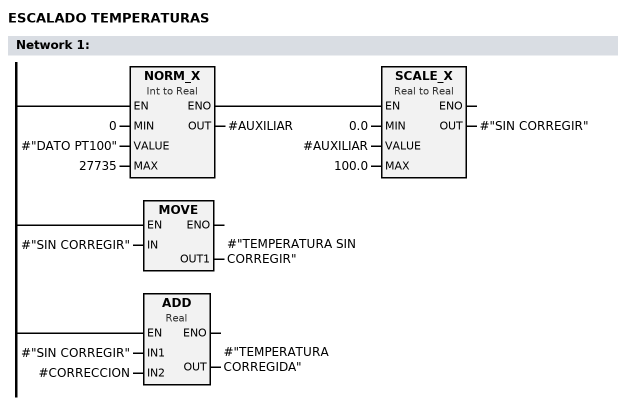
   RUNG wire#powerrail
      { S7_Templates := "[SrcType := Int, DestType := Real]" } Normalize(min := 0, value := #"DATO PT100", max := 27735, out => #AUXILIAR)
      { S7_Templates := "[SrcType := Real, DestType := Real]" } Scale(min := 0.0, value := #AUXILIAR, max := 100.0, out => #"SIN CORREGIR")
   END_RUNG
   RUNG wire#powerrail
      Move(in := #"SIN CORREGIR", out1 => #"TEMPERATURA SIN CORREGIR")
   END_RUNG
   RUNG wire#powerrail
      { S7_Templates := "SrcType := Real" } Add(in1 := #"SIN CORREGIR", in2 := #CORRECCION, out => #"TEMPERATURA CORREGIDA")
   END_RUNG
   // the same network as SCL:
   #AUXILIAR := NORM_X(MIN := 0, VALUE := #"DATO PT100", MAX := 27735);
   #"SIN CORREGIR" := SCALE_X(MIN := 0.0, VALUE := #AUXILIAR, MAX := 100.0);
   #"TEMPERATURA SIN CORREGIR" := #"SIN CORREGIR";
   #"TEMPERATURA CORREGIDA" := #"SIN CORREGIR" + #CORRECCION;
END_REGION
END_FUNCTION

FUNCTION "CONVERSOR MIN A MS" : Void   // FC2, LAD
{ S7_Optimized_Access := 'TRUE' }
VERSION : 0.1
   VAR_INPUT
      "TIEMPO EN MIN" : Int;
   END_VAR
   VAR_OUTPUT
      "TIEMPO EN MS" : DInt;
   END_VAR
BEGIN

REGION Network 1
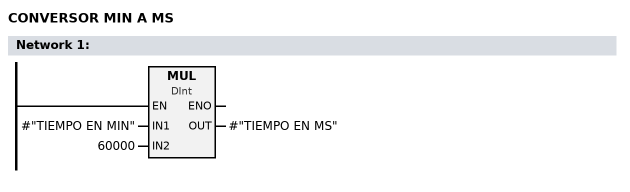
   RUNG wire#powerrail
      { S7_Templates := "SrcType := DInt" } Mul(in1 := #"TIEMPO EN MIN", in2 := 60000, out => #"TIEMPO EN MS")
   END_RUNG
   // the same network as SCL:
   #"TIEMPO EN MS" := #"TIEMPO EN MIN" * 60000;
END_REGION
END_FUNCTION

FUNCTION "CONVERSOR MS A MIN" : Void   // FC3, LAD
{ S7_Optimized_Access := 'TRUE' }
VERSION : 0.1
   VAR_INPUT
      "TIEMPO EN MS" : DInt;
   END_VAR
   VAR_OUTPUT
      "TIEMPO EN MIN" : Int;
   END_VAR
BEGIN

REGION Network 1
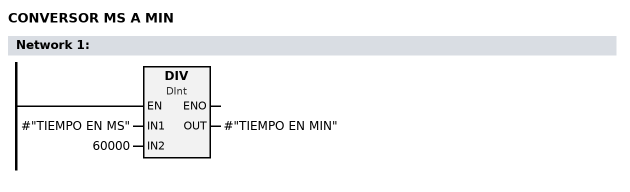
   RUNG wire#powerrail
      { S7_Templates := "SrcType := DInt" } Div(in1 := #"TIEMPO EN MS", in2 := 60000, out => #"TIEMPO EN MIN")
   END_RUNG
   // the same network as SCL:
   #"TIEMPO EN MIN" := #"TIEMPO EN MS" / 60000;
END_REGION
END_FUNCTION

ORGANIZATION_BLOCK "Main"   // OB1, LAD, ProgramCycle
TITLE = "Main Program Sweep (Cycle)"
{ S7_Optimized_Access := 'TRUE' }
VERSION : 0.1
   VAR_INPUT
      Initial_Call : Bool;   // Initial call of this OB
      Remanence : Bool;   // =True, if remanent data are available
   END_VAR
   VAR CONSTANT
      "LARGO REGLA" : Int := 1240;
      COCINA : String := 'COCINA';
      ENFRIADOR : String := 'ENFRIADOR';
   END_VAR
   VAR_TEMP   // added for the SCL form of the ladder/FBD networks
      _w1 : Bool;
   END_VAR
BEGIN

REGION Network 1: REARME
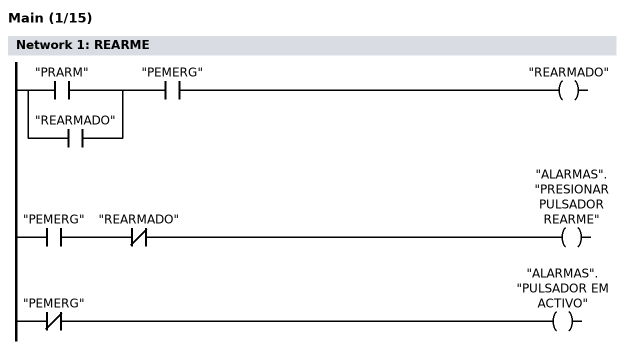
   RUNG wire#powerrail
      Contact( "PRARM" )
      wire#w1
      Contact( "PEMERG" )
      Coil( "REARMADO" )
   END_RUNG
   RUNG wire#powerrail
      Contact( "REARMADO" )
   END_RUNG wire#w1
   RUNG wire#powerrail
      Contact( "PEMERG" )
      I_Contact( "REARMADO" )
      Coil( "ALARMAS"."PRESIONAR PULSADOR REARME" )
   END_RUNG
   RUNG wire#powerrail
      I_Contact( "PEMERG" )
      Coil( "ALARMAS"."PULSADOR EM ACTIVO" )
   END_RUNG
   // the same network as SCL:
   "REARMADO" := ("PRARM" OR "REARMADO") AND "PEMERG";
   "ALARMAS"."PRESIONAR PULSADOR REARME" := "PEMERG" AND NOT "REARMADO";
   "ALARMAS"."PULSADOR EM ACTIVO" := NOT "PEMERG";
END_REGION

REGION Network 2: SELECCION DE NUMERO DE EQUIPO
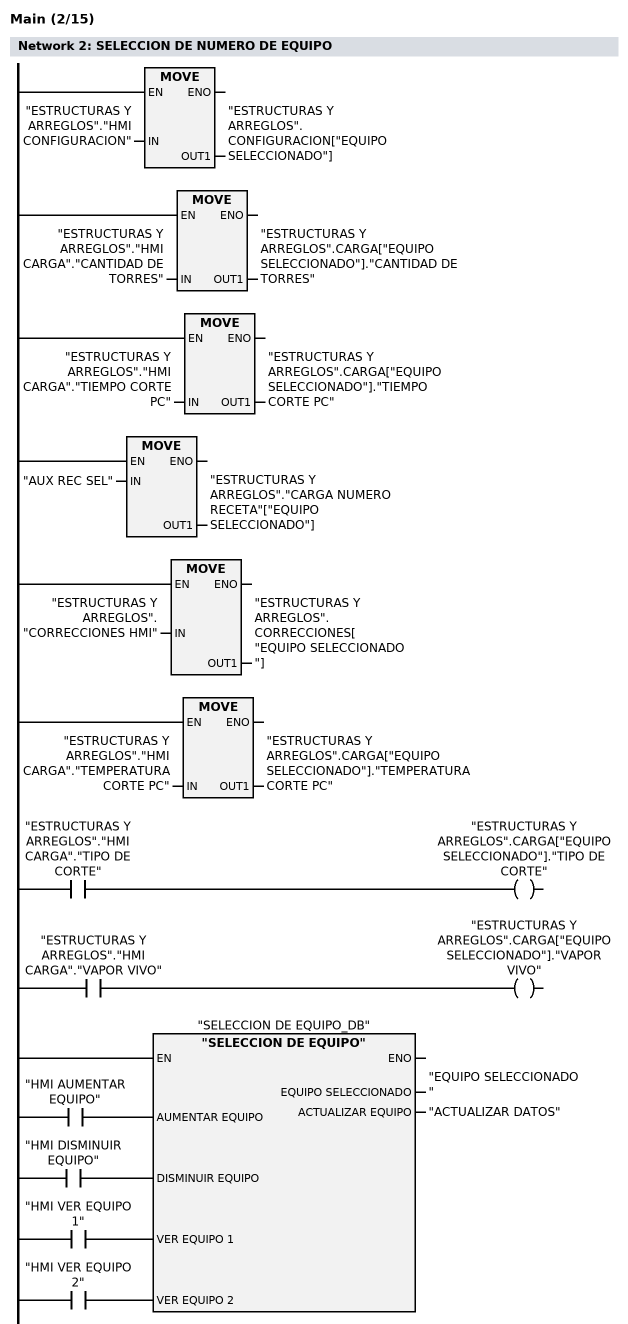
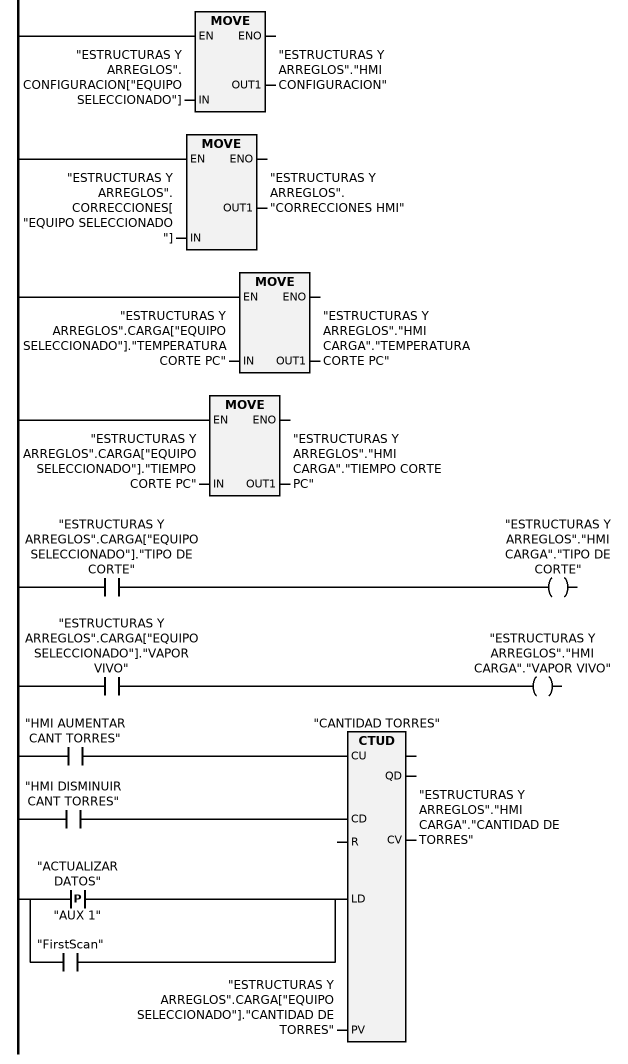
   "ESTRUCTURAS Y ARREGLOS".CONFIGURACION["EQUIPO SELECCIONADO"] := "ESTRUCTURAS Y ARREGLOS"."HMI CONFIGURACION";
   "ESTRUCTURAS Y ARREGLOS".CARGA["EQUIPO SELECCIONADO"]."CANTIDAD DE TORRES" := "ESTRUCTURAS Y ARREGLOS"."HMI CARGA"."CANTIDAD DE TORRES";
   "ESTRUCTURAS Y ARREGLOS".CARGA["EQUIPO SELECCIONADO"]."TIEMPO CORTE PC" := "ESTRUCTURAS Y ARREGLOS"."HMI CARGA"."TIEMPO CORTE PC";
   "ESTRUCTURAS Y ARREGLOS"."CARGA NUMERO RECETA"["EQUIPO SELECCIONADO"] := "AUX REC SEL";
   "ESTRUCTURAS Y ARREGLOS".CORRECCIONES["EQUIPO SELECCIONADO"] := "ESTRUCTURAS Y ARREGLOS"."CORRECCIONES HMI";
   "ESTRUCTURAS Y ARREGLOS".CARGA["EQUIPO SELECCIONADO"]."TEMPERATURA CORTE PC" := "ESTRUCTURAS Y ARREGLOS"."HMI CARGA"."TEMPERATURA CORTE PC";
   "ESTRUCTURAS Y ARREGLOS".CARGA["EQUIPO SELECCIONADO"]."TIPO DE CORTE" := "ESTRUCTURAS Y ARREGLOS"."HMI CARGA"."TIPO DE CORTE";
   "ESTRUCTURAS Y ARREGLOS".CARGA["EQUIPO SELECCIONADO"]."VAPOR VIVO" := "ESTRUCTURAS Y ARREGLOS"."HMI CARGA"."VAPOR VIVO";
   "SELECCION DE EQUIPO_DB"("AUMENTAR EQUIPO" := "HMI AUMENTAR EQUIPO",   // "SELECCION DE EQUIPO"
                           "DISMINUIR EQUIPO" := "HMI DISMINUIR EQUIPO",
                           "VER EQUIPO 1" := "HMI VER EQUIPO 1",
                           "VER EQUIPO 2" := "HMI VER EQUIPO 2",
                           "EQUIPO SELECCIONADO" => "EQUIPO SELECCIONADO",
                           "ACTUALIZAR EQUIPO" => "ACTUALIZAR DATOS");
   "ESTRUCTURAS Y ARREGLOS"."HMI CONFIGURACION" := "ESTRUCTURAS Y ARREGLOS".CONFIGURACION["EQUIPO SELECCIONADO"];
   "ESTRUCTURAS Y ARREGLOS"."CORRECCIONES HMI" := "ESTRUCTURAS Y ARREGLOS".CORRECCIONES["EQUIPO SELECCIONADO"];
   "ESTRUCTURAS Y ARREGLOS"."HMI CARGA"."TEMPERATURA CORTE PC" := "ESTRUCTURAS Y ARREGLOS".CARGA["EQUIPO SELECCIONADO"]."TEMPERATURA CORTE PC";
   "ESTRUCTURAS Y ARREGLOS"."HMI CARGA"."TIEMPO CORTE PC" := "ESTRUCTURAS Y ARREGLOS".CARGA["EQUIPO SELECCIONADO"]."TIEMPO CORTE PC";
   "ESTRUCTURAS Y ARREGLOS"."HMI CARGA"."TIPO DE CORTE" := "ESTRUCTURAS Y ARREGLOS".CARGA["EQUIPO SELECCIONADO"]."TIPO DE CORTE";
   "ESTRUCTURAS Y ARREGLOS"."HMI CARGA"."VAPOR VIVO" := "ESTRUCTURAS Y ARREGLOS".CARGA["EQUIPO SELECCIONADO"]."VAPOR VIVO";
   #_w1 := "ACTUALIZAR DATOS" AND NOT "AUX 1";   // rising edge of "ACTUALIZAR DATOS"
   "AUX 1" := "ACTUALIZAR DATOS";
   "CANTIDAD TORRES".CTUD(CU := "HMI AUMENTAR CANT TORRES",
                          CD := "HMI DISMINUIR CANT TORRES",
                          LD := #_w1 OR "FirstScan",
                          PV := "ESTRUCTURAS Y ARREGLOS".CARGA["EQUIPO SELECCIONADO"]."CANTIDAD DE TORRES",
                          CV => "ESTRUCTURAS Y ARREGLOS"."HMI CARGA"."CANTIDAD DE TORRES");
END_REGION

REGION Network 3: VISUALIZACION LIMITE CANTIDAD DE EQUIPOS Y CANTIDAD DE TORRES
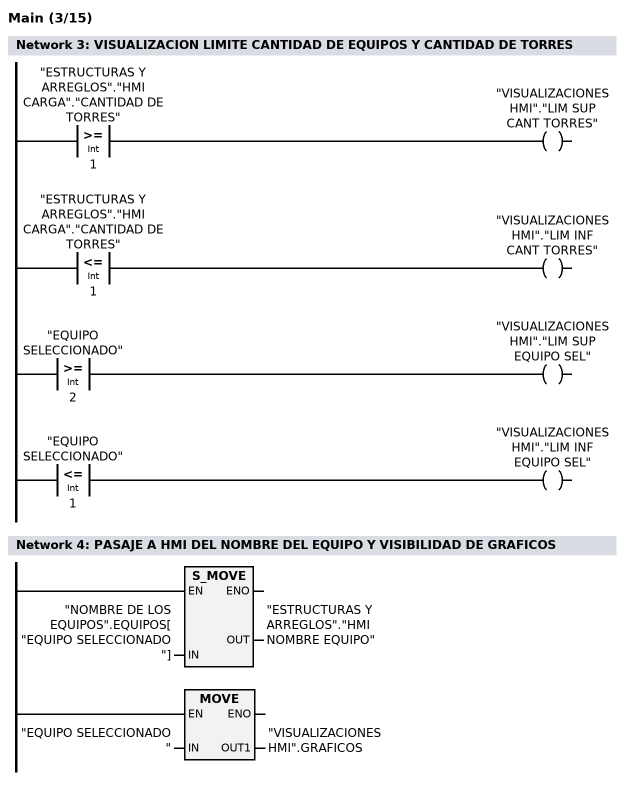
   RUNG wire#powerrail
      { S7_Templates := "SrcType := Int" } GE_Contact(in1 := "ESTRUCTURAS Y ARREGLOS"."HMI CARGA"."CANTIDAD DE TORRES", in2 := 1)
      Coil( "VISUALIZACIONES HMI"."LIM SUP CANT TORRES" )
   END_RUNG
   RUNG wire#powerrail
      { S7_Templates := "SrcType := Int" } LE_Contact(in1 := "ESTRUCTURAS Y ARREGLOS"."HMI CARGA"."CANTIDAD DE TORRES", in2 := 1)
      Coil( "VISUALIZACIONES HMI"."LIM INF CANT TORRES" )
   END_RUNG
   RUNG wire#powerrail
      { S7_Templates := "SrcType := Int" } GE_Contact(in1 := "EQUIPO SELECCIONADO", in2 := 2)
      Coil( "VISUALIZACIONES HMI"."LIM SUP EQUIPO SEL" )
   END_RUNG
   RUNG wire#powerrail
      { S7_Templates := "SrcType := Int" } LE_Contact(in1 := "EQUIPO SELECCIONADO", in2 := 1)
      Coil( "VISUALIZACIONES HMI"."LIM INF EQUIPO SEL" )
   END_RUNG
   // the same network as SCL:
   "VISUALIZACIONES HMI"."LIM SUP CANT TORRES" := "ESTRUCTURAS Y ARREGLOS"."HMI CARGA"."CANTIDAD DE TORRES" >= 1;
   "VISUALIZACIONES HMI"."LIM INF CANT TORRES" := "ESTRUCTURAS Y ARREGLOS"."HMI CARGA"."CANTIDAD DE TORRES" <= 1;
   "VISUALIZACIONES HMI"."LIM SUP EQUIPO SEL" := "EQUIPO SELECCIONADO" >= 2;
   "VISUALIZACIONES HMI"."LIM INF EQUIPO SEL" := "EQUIPO SELECCIONADO" <= 1;
END_REGION

REGION Network 4: PASAJE A HMI DEL NOMBRE DEL EQUIPO Y VISIBILIDAD DE GRAFICOS
   RUNG wire#powerrail
      S_Move(in := "NOMBRE DE LOS EQUIPOS".EQUIPOS["EQUIPO SELECCIONADO"], out => "ESTRUCTURAS Y ARREGLOS"."HMI NOMBRE EQUIPO")
   END_RUNG
   RUNG wire#powerrail
      Move(in := "EQUIPO SELECCIONADO", out1 => "VISUALIZACIONES HMI".GRAFICOS)
   END_RUNG
   // the same network as SCL:
   "ESTRUCTURAS Y ARREGLOS"."HMI NOMBRE EQUIPO" := "NOMBRE DE LOS EQUIPOS".EQUIPOS["EQUIPO SELECCIONADO"];
   "VISUALIZACIONES HMI".GRAFICOS := "EQUIPO SELECCIONADO";
END_REGION

REGION Network 5: BOTON VISUALIZAR RECETA EN PANTALLA "EQUIPO"
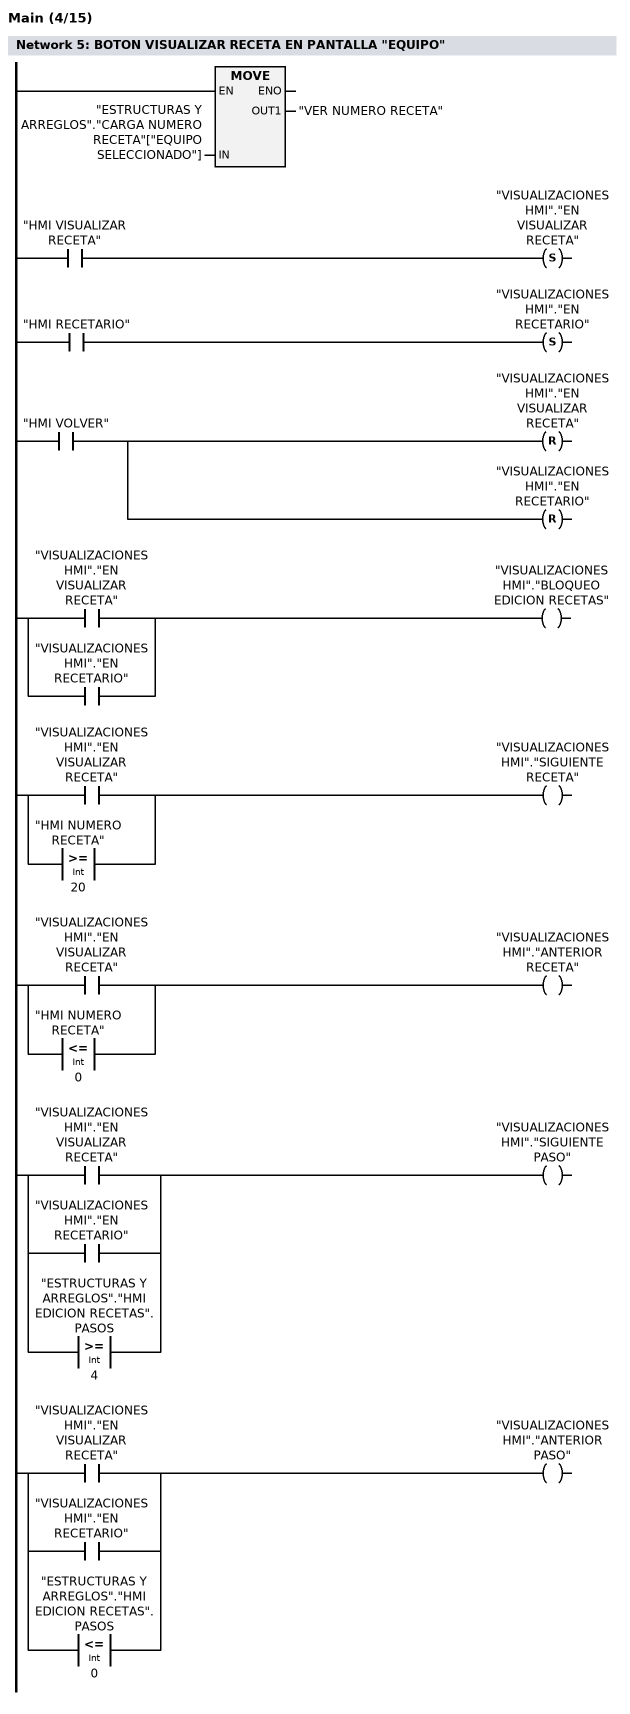
   RUNG wire#powerrail
      Move(in := "ESTRUCTURAS Y ARREGLOS"."CARGA NUMERO RECETA"["EQUIPO SELECCIONADO"], out1 => "VER NUMERO RECETA")
   END_RUNG
   RUNG wire#powerrail
      Contact( "HMI VISUALIZAR RECETA" )
      S_Coil( "VISUALIZACIONES HMI"."EN VISUALIZAR RECETA" )
   END_RUNG
   RUNG wire#powerrail
      Contact( "HMI RECETARIO" )
      S_Coil( "VISUALIZACIONES HMI"."EN RECETARIO" )
   END_RUNG
   RUNG wire#powerrail
      Contact( "HMI VOLVER" )
      wire#w1
      R_Coil( "VISUALIZACIONES HMI"."EN VISUALIZAR RECETA" )
   END_RUNG
   RUNG wire#w1
      R_Coil( "VISUALIZACIONES HMI"."EN RECETARIO" )
   END_RUNG
   RUNG wire#powerrail
      Contact( "VISUALIZACIONES HMI"."EN VISUALIZAR RECETA" )
      wire#w2
      Coil( "VISUALIZACIONES HMI"."BLOQUEO EDICION RECETAS" )
   END_RUNG
   RUNG wire#powerrail
      Contact( "VISUALIZACIONES HMI"."EN RECETARIO" )
   END_RUNG wire#w2
   RUNG wire#powerrail
      Contact( "VISUALIZACIONES HMI"."EN VISUALIZAR RECETA" )
      wire#w3
      Coil( "VISUALIZACIONES HMI"."SIGUIENTE RECETA" )
   END_RUNG
   RUNG wire#powerrail
      { S7_Templates := "SrcType := Int" } GE_Contact(in1 := "HMI NUMERO RECETA", in2 := 20)
   END_RUNG wire#w3
   RUNG wire#powerrail
      Contact( "VISUALIZACIONES HMI"."EN VISUALIZAR RECETA" )
      wire#w4
      Coil( "VISUALIZACIONES HMI"."ANTERIOR RECETA" )
   END_RUNG
   RUNG wire#powerrail
      { S7_Templates := "SrcType := Int" } LE_Contact(in1 := "HMI NUMERO RECETA", in2 := 0)
   END_RUNG wire#w4
   RUNG wire#powerrail
      Contact( "VISUALIZACIONES HMI"."EN VISUALIZAR RECETA" )
      wire#w5
      Coil( "VISUALIZACIONES HMI"."SIGUIENTE PASO" )
   END_RUNG
   RUNG wire#powerrail
      Contact( "VISUALIZACIONES HMI"."EN RECETARIO" )
   END_RUNG wire#w5
   RUNG wire#powerrail
      { S7_Templates := "SrcType := Int" } GE_Contact(in1 := "ESTRUCTURAS Y ARREGLOS"."HMI EDICION RECETAS".PASOS, in2 := 4)
   END_RUNG wire#w5
   RUNG wire#powerrail
      Contact( "VISUALIZACIONES HMI"."EN VISUALIZAR RECETA" )
      wire#w6
      Coil( "VISUALIZACIONES HMI"."ANTERIOR PASO" )
   END_RUNG
   RUNG wire#powerrail
      Contact( "VISUALIZACIONES HMI"."EN RECETARIO" )
   END_RUNG wire#w6
   RUNG wire#powerrail
      { S7_Templates := "SrcType := Int" } LE_Contact(in1 := "ESTRUCTURAS Y ARREGLOS"."HMI EDICION RECETAS".PASOS, in2 := 0)
   END_RUNG wire#w6
   // the same network as SCL:
   "VER NUMERO RECETA" := "ESTRUCTURAS Y ARREGLOS"."CARGA NUMERO RECETA"["EQUIPO SELECCIONADO"];
   IF "HMI VISUALIZAR RECETA" THEN "VISUALIZACIONES HMI"."EN VISUALIZAR RECETA" := TRUE; END_IF;
   IF "HMI RECETARIO" THEN "VISUALIZACIONES HMI"."EN RECETARIO" := TRUE; END_IF;
   IF "HMI VOLVER" THEN
       "VISUALIZACIONES HMI"."EN VISUALIZAR RECETA" := FALSE;
       "VISUALIZACIONES HMI"."EN RECETARIO" := FALSE;
   END_IF;
   "VISUALIZACIONES HMI"."BLOQUEO EDICION RECETAS" := "VISUALIZACIONES HMI"."EN VISUALIZAR RECETA" OR "VISUALIZACIONES HMI"."EN RECETARIO";
   "VISUALIZACIONES HMI"."SIGUIENTE RECETA" := "VISUALIZACIONES HMI"."EN VISUALIZAR RECETA" OR ("HMI NUMERO RECETA" >= 20);
   "VISUALIZACIONES HMI"."ANTERIOR RECETA" := "VISUALIZACIONES HMI"."EN VISUALIZAR RECETA" OR ("HMI NUMERO RECETA" <= 0);
   "VISUALIZACIONES HMI"."SIGUIENTE PASO" := "VISUALIZACIONES HMI"."EN VISUALIZAR RECETA" OR "VISUALIZACIONES HMI"."EN RECETARIO" OR ("ESTRUCTURAS Y ARREGLOS"."HMI EDICION RECETAS".PASOS >= 4);
   "VISUALIZACIONES HMI"."ANTERIOR PASO" := "VISUALIZACIONES HMI"."EN VISUALIZAR RECETA" OR "VISUALIZACIONES HMI"."EN RECETARIO" OR ("ESTRUCTURAS Y ARREGLOS"."HMI EDICION RECETAS".PASOS <= 0);
END_REGION

REGION Network 6: EDITAR RECETAS
   // Receta
   // Recetario
   // Buscar y cargar rece
   // 
   // LOS PASOS TIENE Q IR POR SEPARADOL DE LA ESTRUCTURA
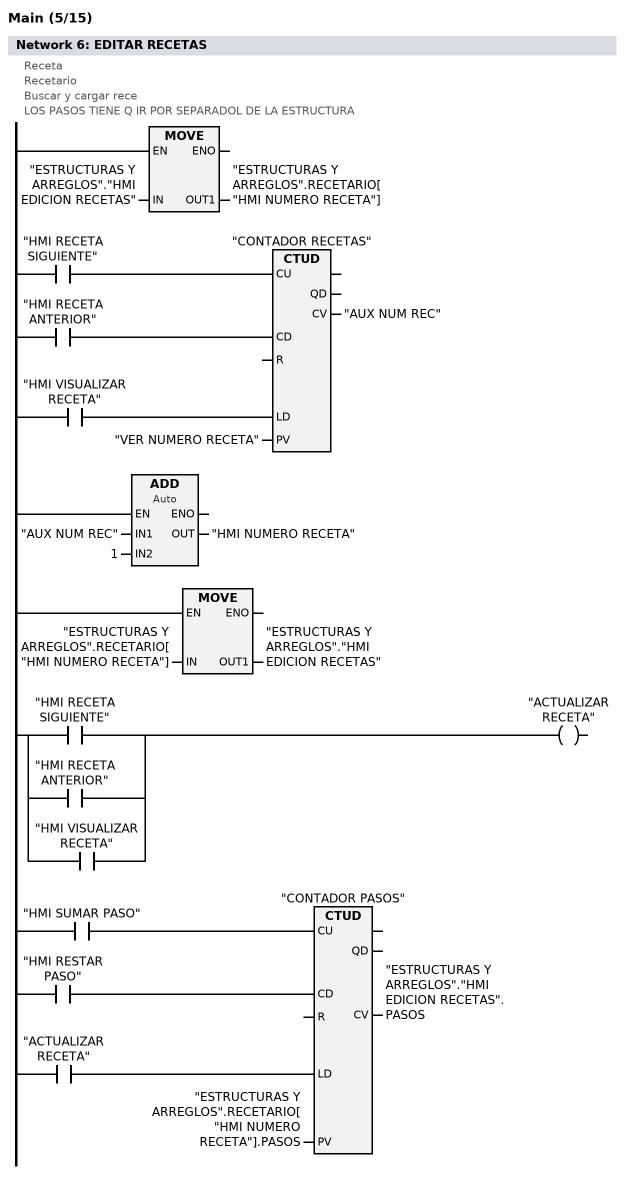
   "ESTRUCTURAS Y ARREGLOS".RECETARIO["HMI NUMERO RECETA"] := "ESTRUCTURAS Y ARREGLOS"."HMI EDICION RECETAS";
   "CONTADOR RECETAS".CTUD(CU := "HMI RECETA SIGUIENTE",
                           CD := "HMI RECETA ANTERIOR",
                           LD := "HMI VISUALIZAR RECETA",
                           PV := "VER NUMERO RECETA",
                           CV => "AUX NUM REC");
   "HMI NUMERO RECETA" := "AUX NUM REC" + 1;
   "ESTRUCTURAS Y ARREGLOS"."HMI EDICION RECETAS" := "ESTRUCTURAS Y ARREGLOS".RECETARIO["HMI NUMERO RECETA"];
   "ACTUALIZAR RECETA" := "HMI RECETA SIGUIENTE" OR "HMI RECETA ANTERIOR" OR "HMI VISUALIZAR RECETA";
   "CONTADOR PASOS".CTUD(CU := "HMI SUMAR PASO",
                         CD := "HMI RESTAR PASO",
                         LD := "ACTUALIZAR RECETA",
                         PV := "ESTRUCTURAS Y ARREGLOS".RECETARIO["HMI NUMERO RECETA"].PASOS,
                         CV => "ESTRUCTURAS Y ARREGLOS"."HMI EDICION RECETAS".PASOS);
END_REGION

REGION Network 7: VISUALIZACIONES RECETA
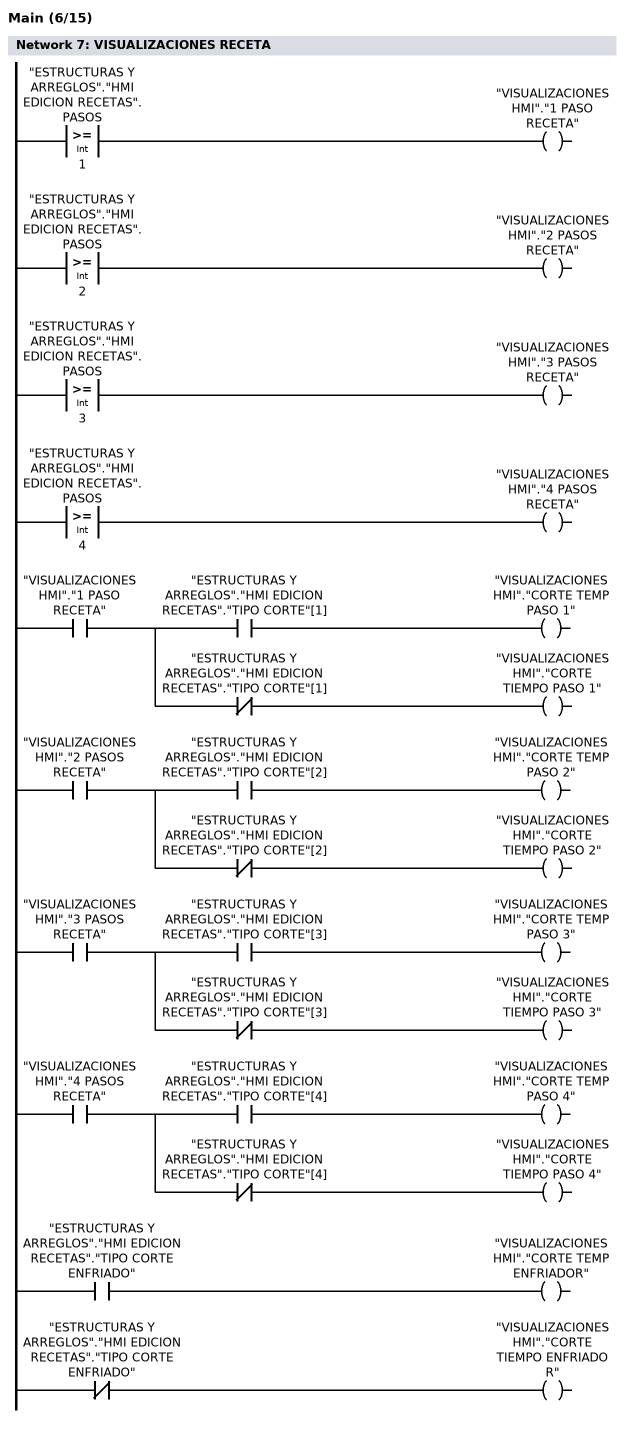
   RUNG wire#powerrail
      { S7_Templates := "SrcType := Int" } GE_Contact(in1 := "ESTRUCTURAS Y ARREGLOS"."HMI EDICION RECETAS".PASOS, in2 := 1)
      Coil( "VISUALIZACIONES HMI"."1 PASO RECETA" )
   END_RUNG
   RUNG wire#powerrail
      { S7_Templates := "SrcType := Int" } GE_Contact(in1 := "ESTRUCTURAS Y ARREGLOS"."HMI EDICION RECETAS".PASOS, in2 := 2)
      Coil( "VISUALIZACIONES HMI"."2 PASOS RECETA" )
   END_RUNG
   RUNG wire#powerrail
      { S7_Templates := "SrcType := Int" } GE_Contact(in1 := "ESTRUCTURAS Y ARREGLOS"."HMI EDICION RECETAS".PASOS, in2 := 3)
      Coil( "VISUALIZACIONES HMI"."3 PASOS RECETA" )
   END_RUNG
   RUNG wire#powerrail
      { S7_Templates := "SrcType := Int" } GE_Contact(in1 := "ESTRUCTURAS Y ARREGLOS"."HMI EDICION RECETAS".PASOS, in2 := 4)
      Coil( "VISUALIZACIONES HMI"."4 PASOS RECETA" )
   END_RUNG
   RUNG wire#powerrail
      Contact( "VISUALIZACIONES HMI"."1 PASO RECETA" )
      wire#w1
      Contact( "ESTRUCTURAS Y ARREGLOS"."HMI EDICION RECETAS"."TIPO CORTE"[1] )
      Coil( "VISUALIZACIONES HMI"."CORTE TEMP PASO 1" )
   END_RUNG
   RUNG wire#w1
      I_Contact( "ESTRUCTURAS Y ARREGLOS"."HMI EDICION RECETAS"."TIPO CORTE"[1] )
      Coil( "VISUALIZACIONES HMI"."CORTE TIEMPO PASO 1" )
   END_RUNG
   RUNG wire#powerrail
      Contact( "VISUALIZACIONES HMI"."2 PASOS RECETA" )
      wire#w2
      Contact( "ESTRUCTURAS Y ARREGLOS"."HMI EDICION RECETAS"."TIPO CORTE"[2] )
      Coil( "VISUALIZACIONES HMI"."CORTE TEMP PASO 2" )
   END_RUNG
   RUNG wire#w2
      I_Contact( "ESTRUCTURAS Y ARREGLOS"."HMI EDICION RECETAS"."TIPO CORTE"[2] )
      Coil( "VISUALIZACIONES HMI"."CORTE TIEMPO PASO 2" )
   END_RUNG
   RUNG wire#powerrail
      Contact( "VISUALIZACIONES HMI"."3 PASOS RECETA" )
      wire#w3
      Contact( "ESTRUCTURAS Y ARREGLOS"."HMI EDICION RECETAS"."TIPO CORTE"[3] )
      Coil( "VISUALIZACIONES HMI"."CORTE TEMP PASO 3" )
   END_RUNG
   RUNG wire#w3
      I_Contact( "ESTRUCTURAS Y ARREGLOS"."HMI EDICION RECETAS"."TIPO CORTE"[3] )
      Coil( "VISUALIZACIONES HMI"."CORTE TIEMPO PASO 3" )
   END_RUNG
   RUNG wire#powerrail
      Contact( "VISUALIZACIONES HMI"."4 PASOS RECETA" )
      wire#w4
      Contact( "ESTRUCTURAS Y ARREGLOS"."HMI EDICION RECETAS"."TIPO CORTE"[4] )
      Coil( "VISUALIZACIONES HMI"."CORTE TEMP PASO 4" )
   END_RUNG
   RUNG wire#w4
      I_Contact( "ESTRUCTURAS Y ARREGLOS"."HMI EDICION RECETAS"."TIPO CORTE"[4] )
      Coil( "VISUALIZACIONES HMI"."CORTE TIEMPO PASO 4" )
   END_RUNG
   RUNG wire#powerrail
      Contact( "ESTRUCTURAS Y ARREGLOS"."HMI EDICION RECETAS"."TIPO CORTE ENFRIADO" )
      Coil( "VISUALIZACIONES HMI"."CORTE TEMP ENFRIADOR" )
   END_RUNG
   RUNG wire#powerrail
      I_Contact( "ESTRUCTURAS Y ARREGLOS"."HMI EDICION RECETAS"."TIPO CORTE ENFRIADO" )
      Coil( "VISUALIZACIONES HMI"."CORTE TIEMPO ENFRIADOR" )
   END_RUNG
   // the same network as SCL:
   "VISUALIZACIONES HMI"."1 PASO RECETA" := "ESTRUCTURAS Y ARREGLOS"."HMI EDICION RECETAS".PASOS >= 1;
   "VISUALIZACIONES HMI"."2 PASOS RECETA" := "ESTRUCTURAS Y ARREGLOS"."HMI EDICION RECETAS".PASOS >= 2;
   "VISUALIZACIONES HMI"."3 PASOS RECETA" := "ESTRUCTURAS Y ARREGLOS"."HMI EDICION RECETAS".PASOS >= 3;
   "VISUALIZACIONES HMI"."4 PASOS RECETA" := "ESTRUCTURAS Y ARREGLOS"."HMI EDICION RECETAS".PASOS >= 4;
   "VISUALIZACIONES HMI"."CORTE TEMP PASO 1" := "VISUALIZACIONES HMI"."1 PASO RECETA" AND "ESTRUCTURAS Y ARREGLOS"."HMI EDICION RECETAS"."TIPO CORTE"[1];
   "VISUALIZACIONES HMI"."CORTE TIEMPO PASO 1" := "VISUALIZACIONES HMI"."1 PASO RECETA" AND NOT "ESTRUCTURAS Y ARREGLOS"."HMI EDICION RECETAS"."TIPO CORTE"[1];
   "VISUALIZACIONES HMI"."CORTE TEMP PASO 2" := "VISUALIZACIONES HMI"."2 PASOS RECETA" AND "ESTRUCTURAS Y ARREGLOS"."HMI EDICION RECETAS"."TIPO CORTE"[2];
   "VISUALIZACIONES HMI"."CORTE TIEMPO PASO 2" := "VISUALIZACIONES HMI"."2 PASOS RECETA" AND NOT "ESTRUCTURAS Y ARREGLOS"."HMI EDICION RECETAS"."TIPO CORTE"[2];
   "VISUALIZACIONES HMI"."CORTE TEMP PASO 3" := "VISUALIZACIONES HMI"."3 PASOS RECETA" AND "ESTRUCTURAS Y ARREGLOS"."HMI EDICION RECETAS"."TIPO CORTE"[3];
   "VISUALIZACIONES HMI"."CORTE TIEMPO PASO 3" := "VISUALIZACIONES HMI"."3 PASOS RECETA" AND NOT "ESTRUCTURAS Y ARREGLOS"."HMI EDICION RECETAS"."TIPO CORTE"[3];
   "VISUALIZACIONES HMI"."CORTE TEMP PASO 4" := "VISUALIZACIONES HMI"."4 PASOS RECETA" AND "ESTRUCTURAS Y ARREGLOS"."HMI EDICION RECETAS"."TIPO CORTE"[4];
   "VISUALIZACIONES HMI"."CORTE TIEMPO PASO 4" := "VISUALIZACIONES HMI"."4 PASOS RECETA" AND NOT "ESTRUCTURAS Y ARREGLOS"."HMI EDICION RECETAS"."TIPO CORTE"[4];
   "VISUALIZACIONES HMI"."CORTE TEMP ENFRIADOR" := "ESTRUCTURAS Y ARREGLOS"."HMI EDICION RECETAS"."TIPO CORTE ENFRIADO";
   "VISUALIZACIONES HMI"."CORTE TIEMPO ENFRIADOR" := NOT "ESTRUCTURAS Y ARREGLOS"."HMI EDICION RECETAS"."TIPO CORTE ENFRIADO";
END_REGION

REGION Network 8: ELEGIR RECETA
   // El comando de PV esta arriba de la funcion contador de equipo
   // 
   // El ultimo Move pasa la receta (del recetario) al equipo seleccionado (1....4) por lo que ya tengo la receta( 1.....20)  almacenada en cada equipo.
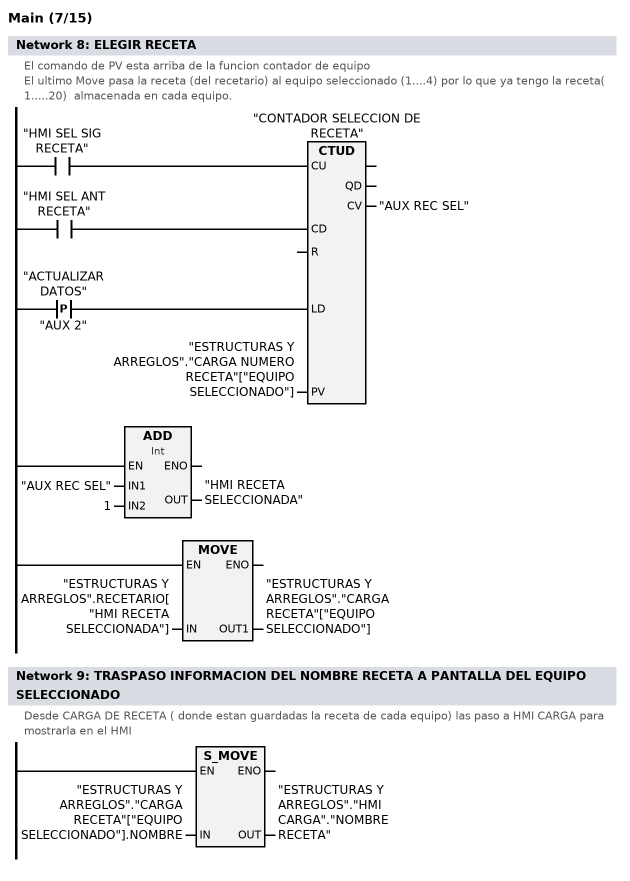
   #_w1 := "ACTUALIZAR DATOS" AND NOT "AUX 2";   // rising edge of "ACTUALIZAR DATOS"
   "AUX 2" := "ACTUALIZAR DATOS";
   "CONTADOR SELECCION DE RECETA".CTUD(CU := "HMI SEL SIG RECETA",
                           CD := "HMI SEL ANT RECETA",
                           LD := #_w1,
                           PV := "ESTRUCTURAS Y ARREGLOS"."CARGA NUMERO RECETA"["EQUIPO SELECCIONADO"],
                           CV => "AUX REC SEL");
   "HMI RECETA SELECCIONADA" := "AUX REC SEL" + 1;
   "ESTRUCTURAS Y ARREGLOS"."CARGA RECETA"["EQUIPO SELECCIONADO"] := "ESTRUCTURAS Y ARREGLOS".RECETARIO["HMI RECETA SELECCIONADA"];
END_REGION

REGION Network 9: TRASPASO INFORMACION DEL NOMBRE RECETA A PANTALLA DEL EQUIPO SELECCIONADO
   // Desde CARGA DE RECETA ( donde estan guardadas la receta de cada equipo) las paso a HMI CARGA para mostrarla en el HMI
   RUNG wire#powerrail
      S_Move(in := "ESTRUCTURAS Y ARREGLOS"."CARGA RECETA"["EQUIPO SELECCIONADO"].NOMBRE, out => "ESTRUCTURAS Y ARREGLOS"."HMI CARGA"."NOMBRE RECETA")
   END_RUNG
   // the same network as SCL:
   "ESTRUCTURAS Y ARREGLOS"."HMI CARGA"."NOMBRE RECETA" := "ESTRUCTURAS Y ARREGLOS"."CARGA RECETA"["EQUIPO SELECCIONADO"].NOMBRE;
END_REGION

REGION Network 10: CONVERSION TEMPERATURAS Y NIVELES
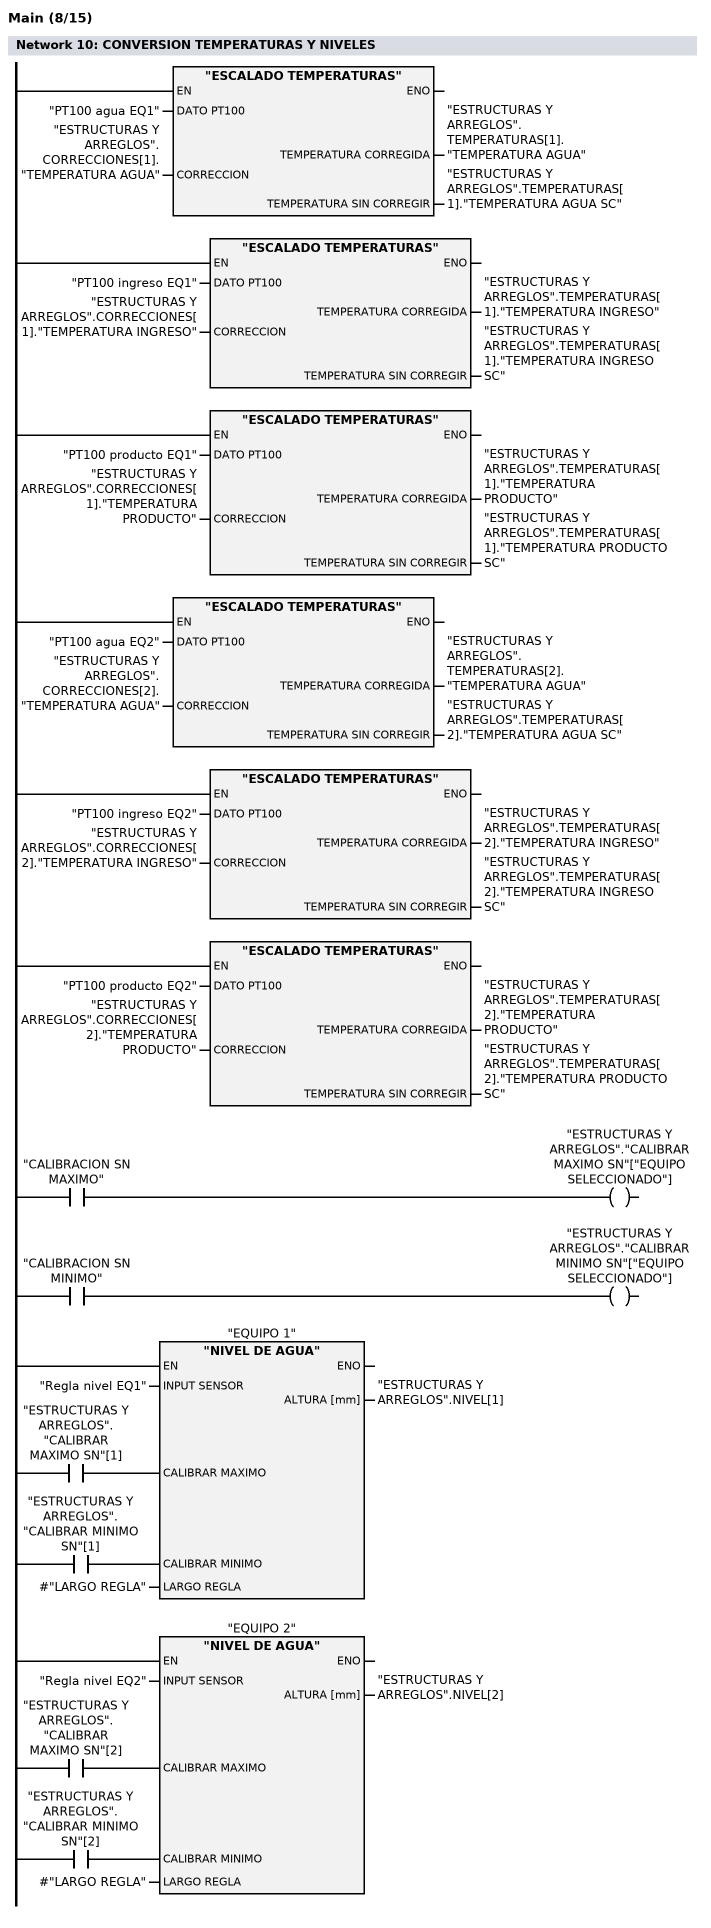
   RUNG wire#powerrail
      "ESCALADO TEMPERATURAS"("DATO PT100" := "PT100 agua EQ1", CORRECCION := "ESTRUCTURAS Y ARREGLOS".CORRECCIONES[1]."TEMPERATURA AGUA", "TEMPERATURA CORREGIDA" => "ESTRUCTURAS Y ARREGLOS".TEMPERATURAS[1]."TEMPERATURA AGUA", "TEMPERATURA SIN CORREGIR" => "ESTRUCTURAS Y ARREGLOS".TEMPERATURAS[1]."TEMPERATURA AGUA SC")
   END_RUNG
   RUNG wire#powerrail
      "ESCALADO TEMPERATURAS"("DATO PT100" := "PT100 ingreso EQ1", CORRECCION := "ESTRUCTURAS Y ARREGLOS".CORRECCIONES[1]."TEMPERATURA INGRESO", "TEMPERATURA CORREGIDA" => "ESTRUCTURAS Y ARREGLOS".TEMPERATURAS[1]."TEMPERATURA INGRESO", "TEMPERATURA SIN CORREGIR" => "ESTRUCTURAS Y ARREGLOS".TEMPERATURAS[1]."TEMPERATURA INGRESO SC")
   END_RUNG
   RUNG wire#powerrail
      "ESCALADO TEMPERATURAS"("DATO PT100" := "PT100 producto EQ1", CORRECCION := "ESTRUCTURAS Y ARREGLOS".CORRECCIONES[1]."TEMPERATURA PRODUCTO", "TEMPERATURA CORREGIDA" => "ESTRUCTURAS Y ARREGLOS".TEMPERATURAS[1]."TEMPERATURA PRODUCTO", "TEMPERATURA SIN CORREGIR" => "ESTRUCTURAS Y ARREGLOS".TEMPERATURAS[1]."TEMPERATURA PRODUCTO SC")
   END_RUNG
   RUNG wire#powerrail
      "ESCALADO TEMPERATURAS"("DATO PT100" := "PT100 agua EQ2", CORRECCION := "ESTRUCTURAS Y ARREGLOS".CORRECCIONES[2]."TEMPERATURA AGUA", "TEMPERATURA CORREGIDA" => "ESTRUCTURAS Y ARREGLOS".TEMPERATURAS[2]."TEMPERATURA AGUA", "TEMPERATURA SIN CORREGIR" => "ESTRUCTURAS Y ARREGLOS".TEMPERATURAS[2]."TEMPERATURA AGUA SC")
   END_RUNG
   RUNG wire#powerrail
      "ESCALADO TEMPERATURAS"("DATO PT100" := "PT100 ingreso EQ2", CORRECCION := "ESTRUCTURAS Y ARREGLOS".CORRECCIONES[2]."TEMPERATURA INGRESO", "TEMPERATURA CORREGIDA" => "ESTRUCTURAS Y ARREGLOS".TEMPERATURAS[2]."TEMPERATURA INGRESO", "TEMPERATURA SIN CORREGIR" => "ESTRUCTURAS Y ARREGLOS".TEMPERATURAS[2]."TEMPERATURA INGRESO SC")
   END_RUNG
   RUNG wire#powerrail
      "ESCALADO TEMPERATURAS"("DATO PT100" := "PT100 producto EQ2", CORRECCION := "ESTRUCTURAS Y ARREGLOS".CORRECCIONES[2]."TEMPERATURA PRODUCTO", "TEMPERATURA CORREGIDA" => "ESTRUCTURAS Y ARREGLOS".TEMPERATURAS[2]."TEMPERATURA PRODUCTO", "TEMPERATURA SIN CORREGIR" => "ESTRUCTURAS Y ARREGLOS".TEMPERATURAS[2]."TEMPERATURA PRODUCTO SC")
   END_RUNG
   RUNG wire#powerrail
      Contact( "CALIBRACION SN MAXIMO" )
      Coil( "ESTRUCTURAS Y ARREGLOS"."CALIBRAR MAXIMO SN"["EQUIPO SELECCIONADO"] )
   END_RUNG
   RUNG wire#powerrail
      Contact( "CALIBRACION SN MINIMO" )
      Coil( "ESTRUCTURAS Y ARREGLOS"."CALIBRAR MINIMO SN"["EQUIPO SELECCIONADO"] )
   END_RUNG
   RUNG wire#powerrail
      "EQUIPO 1"("CALIBRAR MAXIMO" := wire#w1, "CALIBRAR MINIMO" := wire#w2, "INPUT SENSOR" := "Regla nivel EQ1", "LARGO REGLA" := #"LARGO REGLA", "ALTURA [mm]" => "ESTRUCTURAS Y ARREGLOS".NIVEL[1])
   END_RUNG
   RUNG wire#powerrail
      Contact( "ESTRUCTURAS Y ARREGLOS"."CALIBRAR MAXIMO SN"[1] )
   END_RUNG wire#w1
   RUNG wire#powerrail
      Contact( "ESTRUCTURAS Y ARREGLOS"."CALIBRAR MINIMO SN"[1] )
   END_RUNG wire#w2
   RUNG wire#powerrail
      "EQUIPO 2"("CALIBRAR MAXIMO" := wire#w3, "CALIBRAR MINIMO" := wire#w4, "INPUT SENSOR" := "Regla nivel EQ2", "LARGO REGLA" := #"LARGO REGLA", "ALTURA [mm]" => "ESTRUCTURAS Y ARREGLOS".NIVEL[2])
   END_RUNG
   RUNG wire#powerrail
      Contact( "ESTRUCTURAS Y ARREGLOS"."CALIBRAR MAXIMO SN"[2] )
   END_RUNG wire#w3
   RUNG wire#powerrail
      Contact( "ESTRUCTURAS Y ARREGLOS"."CALIBRAR MINIMO SN"[2] )
   END_RUNG wire#w4
   // the same network as SCL:
   "ESCALADO TEMPERATURAS"("DATO PT100" := "PT100 agua EQ1",
                           CORRECCION := "ESTRUCTURAS Y ARREGLOS".CORRECCIONES[1]."TEMPERATURA AGUA",
                           "TEMPERATURA CORREGIDA" => "ESTRUCTURAS Y ARREGLOS".TEMPERATURAS[1]."TEMPERATURA AGUA",
                           "TEMPERATURA SIN CORREGIR" => "ESTRUCTURAS Y ARREGLOS".TEMPERATURAS[1]."TEMPERATURA AGUA SC");
   "ESCALADO TEMPERATURAS"("DATO PT100" := "PT100 ingreso EQ1",
                           CORRECCION := "ESTRUCTURAS Y ARREGLOS".CORRECCIONES[1]."TEMPERATURA INGRESO",
                           "TEMPERATURA CORREGIDA" => "ESTRUCTURAS Y ARREGLOS".TEMPERATURAS[1]."TEMPERATURA INGRESO",
                           "TEMPERATURA SIN CORREGIR" => "ESTRUCTURAS Y ARREGLOS".TEMPERATURAS[1]."TEMPERATURA INGRESO SC");
   "ESCALADO TEMPERATURAS"("DATO PT100" := "PT100 producto EQ1",
                           CORRECCION := "ESTRUCTURAS Y ARREGLOS".CORRECCIONES[1]."TEMPERATURA PRODUCTO",
                           "TEMPERATURA CORREGIDA" => "ESTRUCTURAS Y ARREGLOS".TEMPERATURAS[1]."TEMPERATURA PRODUCTO",
                           "TEMPERATURA SIN CORREGIR" => "ESTRUCTURAS Y ARREGLOS".TEMPERATURAS[1]."TEMPERATURA PRODUCTO SC");
   "ESCALADO TEMPERATURAS"("DATO PT100" := "PT100 agua EQ2",
                           CORRECCION := "ESTRUCTURAS Y ARREGLOS".CORRECCIONES[2]."TEMPERATURA AGUA",
                           "TEMPERATURA CORREGIDA" => "ESTRUCTURAS Y ARREGLOS".TEMPERATURAS[2]."TEMPERATURA AGUA",
                           "TEMPERATURA SIN CORREGIR" => "ESTRUCTURAS Y ARREGLOS".TEMPERATURAS[2]."TEMPERATURA AGUA SC");
   "ESCALADO TEMPERATURAS"("DATO PT100" := "PT100 ingreso EQ2",
                           CORRECCION := "ESTRUCTURAS Y ARREGLOS".CORRECCIONES[2]."TEMPERATURA INGRESO",
                           "TEMPERATURA CORREGIDA" => "ESTRUCTURAS Y ARREGLOS".TEMPERATURAS[2]."TEMPERATURA INGRESO",
                           "TEMPERATURA SIN CORREGIR" => "ESTRUCTURAS Y ARREGLOS".TEMPERATURAS[2]."TEMPERATURA INGRESO SC");
   "ESCALADO TEMPERATURAS"("DATO PT100" := "PT100 producto EQ2",
                           CORRECCION := "ESTRUCTURAS Y ARREGLOS".CORRECCIONES[2]."TEMPERATURA PRODUCTO",
                           "TEMPERATURA CORREGIDA" => "ESTRUCTURAS Y ARREGLOS".TEMPERATURAS[2]."TEMPERATURA PRODUCTO",
                           "TEMPERATURA SIN CORREGIR" => "ESTRUCTURAS Y ARREGLOS".TEMPERATURAS[2]."TEMPERATURA PRODUCTO SC");
   "ESTRUCTURAS Y ARREGLOS"."CALIBRAR MAXIMO SN"["EQUIPO SELECCIONADO"] := "CALIBRACION SN MAXIMO";
   "ESTRUCTURAS Y ARREGLOS"."CALIBRAR MINIMO SN"["EQUIPO SELECCIONADO"] := "CALIBRACION SN MINIMO";
   "EQUIPO 1"("INPUT SENSOR" := "Regla nivel EQ1",   // "NIVEL DE AGUA"
              "CALIBRAR MAXIMO" := "ESTRUCTURAS Y ARREGLOS"."CALIBRAR MAXIMO SN"[1],
              "CALIBRAR MINIMO" := "ESTRUCTURAS Y ARREGLOS"."CALIBRAR MINIMO SN"[1],
              "LARGO REGLA" := #"LARGO REGLA",
              "ALTURA [mm]" => "ESTRUCTURAS Y ARREGLOS".NIVEL[1]);
   "EQUIPO 2"("INPUT SENSOR" := "Regla nivel EQ2",   // "NIVEL DE AGUA"
              "CALIBRAR MAXIMO" := "ESTRUCTURAS Y ARREGLOS"."CALIBRAR MAXIMO SN"[2],
              "CALIBRAR MINIMO" := "ESTRUCTURAS Y ARREGLOS"."CALIBRAR MINIMO SN"[2],
              "LARGO REGLA" := #"LARGO REGLA",
              "ALTURA [mm]" => "ESTRUCTURAS Y ARREGLOS".NIVEL[2]);
END_REGION

REGION Network 11: TRASPASO DE TEMPERATURAS Y NIVELES
   // 1 MOVE : Traspaso de temperaturas a HMI mientras va cambiando el numero de equipo
   // 2 MOVE : Traspaso de correcciones a HMI (en configuraciones) mientras va cambiando el numero de equipo
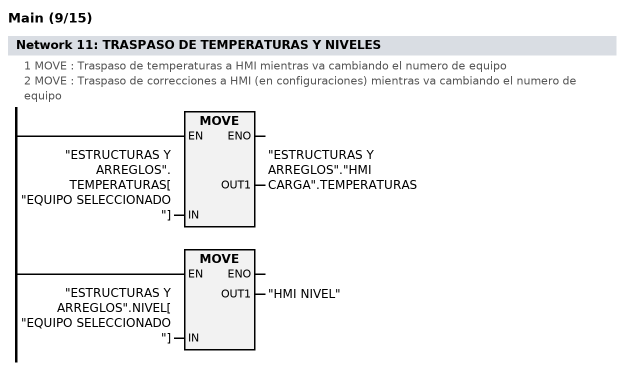
   RUNG wire#powerrail
      Move(in := "ESTRUCTURAS Y ARREGLOS".TEMPERATURAS["EQUIPO SELECCIONADO"], out1 => "ESTRUCTURAS Y ARREGLOS"."HMI CARGA".TEMPERATURAS)
   END_RUNG
   RUNG wire#powerrail
      Move(in := "ESTRUCTURAS Y ARREGLOS".NIVEL["EQUIPO SELECCIONADO"], out1 => "HMI NIVEL")
   END_RUNG
   // the same network as SCL:
   "ESTRUCTURAS Y ARREGLOS"."HMI CARGA".TEMPERATURAS := "ESTRUCTURAS Y ARREGLOS".TEMPERATURAS["EQUIPO SELECCIONADO"];
   "HMI NIVEL" := "ESTRUCTURAS Y ARREGLOS".NIVEL["EQUIPO SELECCIONADO"];
END_REGION

REGION Network 12: EQUIPO 1
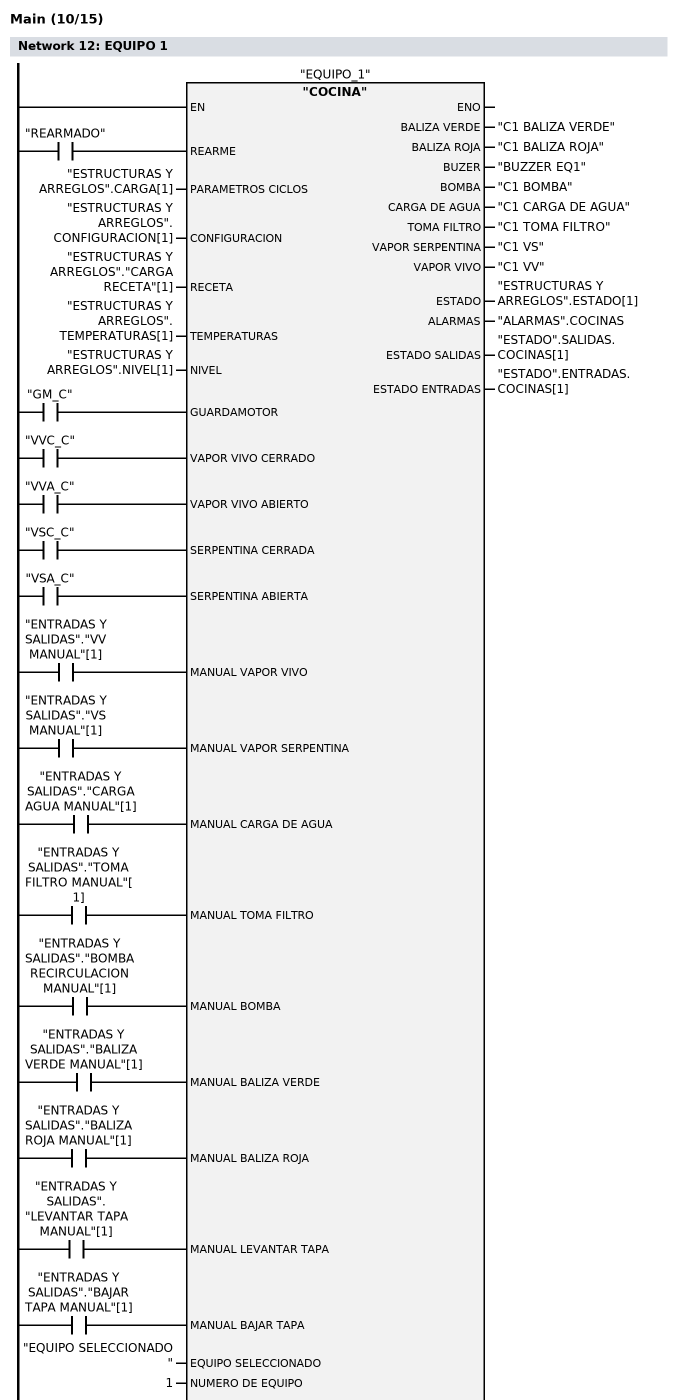
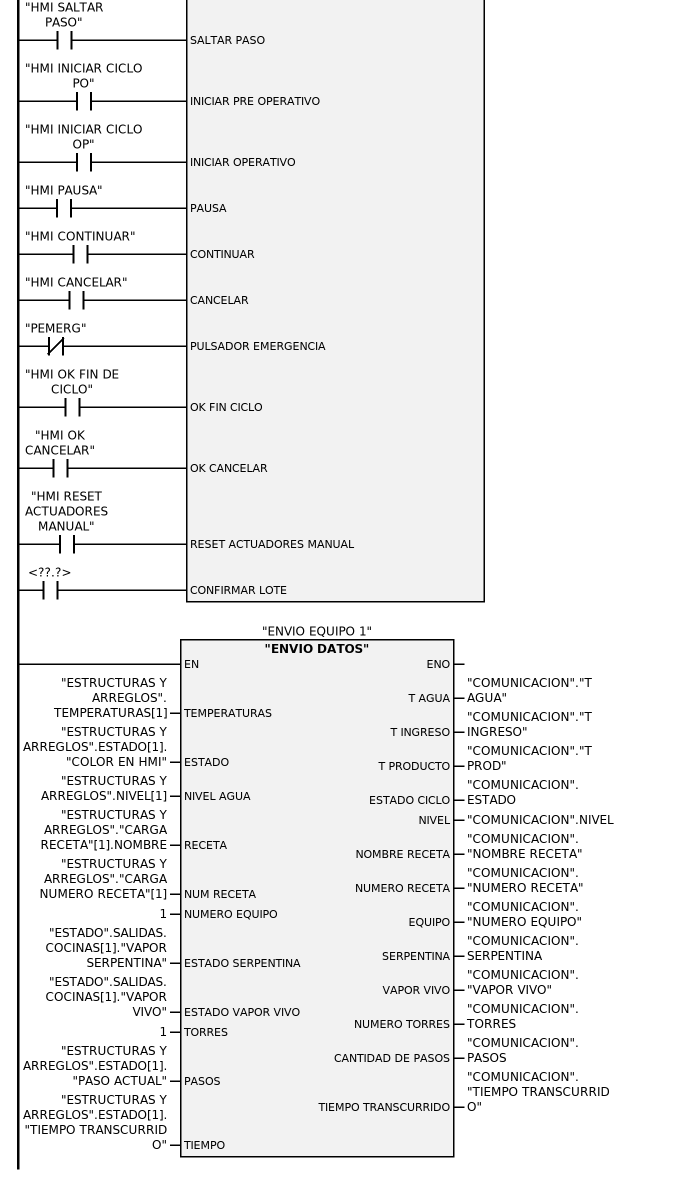
   RUNG wire#powerrail
      "EQUIPO_1"(REARME := wire#w1, GUARDAMOTOR := wire#w2, "VAPOR VIVO CERRADO" := wire#w3, "VAPOR VIVO ABIERTO" := wire#w4, "SERPENTINA CERRADA" := wire#w5, "SERPENTINA ABIERTA" := wire#w6, "MANUAL VAPOR VIVO" := wire#w7, "MANUAL VAPOR SERPENTINA" := wire#w8, "MANUAL CARGA DE AGUA" := wire#w9, "MANUAL TOMA FILTRO" := wire#w10, "MANUAL BOMBA" := wire#w11, "MANUAL BALIZA VERDE" := wire#w12, "MANUAL BALIZA ROJA" := wire#w13, "MANUAL LEVANTAR TAPA" := wire#w14, "MANUAL BAJAR TAPA" := wire#w15, "SALTAR PASO" := wire#w16, "INICIAR PRE OPERATIVO" := wire#w17, "INICIAR OPERATIVO" := wire#w18, PAUSA := wire#w19, CONTINUAR := wire#w20, CANCELAR := wire#w21, "PULSADOR EMERGENCIA" := wire#w22, "OK FIN CICLO" := wire#w23, "OK CANCELAR" := wire#w24, "RESET ACTUADORES MANUAL" := wire#w25, "CONFIRMAR LOTE" := wire#w26, "PARAMETROS CICLOS" := "ESTRUCTURAS Y ARREGLOS".CARGA[1], CONFIGURACION := "ESTRUCTURAS Y ARREGLOS".CONFIGURACION[1], RECETA := "ESTRUCTURAS Y ARREGLOS"."CARGA RECETA"[1], TEMPERATURAS := "ESTRUCTURAS Y ARREGLOS".TEMPERATURAS[1], NIVEL := "ESTRUCTURAS Y ARREGLOS".NIVEL[1], "EQUIPO SELECCIONADO" := "EQUIPO SELECCIONADO", "NUMERO DE EQUIPO" := 1, "BALIZA VERDE" => "C1 BALIZA VERDE", "BALIZA ROJA" => "C1 BALIZA ROJA", BUZER => "BUZZER EQ1", BOMBA => "C1 BOMBA", "CARGA DE AGUA" => "C1 CARGA DE AGUA", "TOMA FILTRO" => "C1 TOMA FILTRO", "VAPOR SERPENTINA" => "C1 VS", "VAPOR VIVO" => "C1 VV", ESTADO => "ESTRUCTURAS Y ARREGLOS".ESTADO[1], ALARMAS => "ALARMAS".COCINAS, "ESTADO SALIDAS" => "ESTADO".SALIDAS.COCINAS[1], "ESTADO ENTRADAS" => "ESTADO".ENTRADAS.COCINAS[1])
   END_RUNG
   RUNG wire#powerrail
      Contact( "REARMADO" )
   END_RUNG wire#w1
   RUNG wire#powerrail
      Contact( "GM_C" )
   END_RUNG wire#w2
   RUNG wire#powerrail
      Contact( "VVC_C" )
   END_RUNG wire#w3
   RUNG wire#powerrail
      Contact( "VVA_C" )
   END_RUNG wire#w4
   RUNG wire#powerrail
      Contact( "VSC_C" )
   END_RUNG wire#w5
   RUNG wire#powerrail
      Contact( "VSA_C" )
   END_RUNG wire#w6
   RUNG wire#powerrail
      Contact( "ENTRADAS Y SALIDAS"."VV MANUAL"[1] )
   END_RUNG wire#w7
   RUNG wire#powerrail
      Contact( "ENTRADAS Y SALIDAS"."VS MANUAL"[1] )
   END_RUNG wire#w8
   RUNG wire#powerrail
      Contact( "ENTRADAS Y SALIDAS"."CARGA AGUA MANUAL"[1] )
   END_RUNG wire#w9
   RUNG wire#powerrail
      Contact( "ENTRADAS Y SALIDAS"."TOMA FILTRO MANUAL"[1] )
   END_RUNG wire#w10
   RUNG wire#powerrail
      Contact( "ENTRADAS Y SALIDAS"."BOMBA RECIRCULACION MANUAL"[1] )
   END_RUNG wire#w11
   RUNG wire#powerrail
      Contact( "ENTRADAS Y SALIDAS"."BALIZA VERDE MANUAL"[1] )
   END_RUNG wire#w12
   RUNG wire#powerrail
      Contact( "ENTRADAS Y SALIDAS"."BALIZA ROJA MANUAL"[1] )
   END_RUNG wire#w13
   RUNG wire#powerrail
      Contact( "ENTRADAS Y SALIDAS"."LEVANTAR TAPA MANUAL"[1] )
   END_RUNG wire#w14
   RUNG wire#powerrail
      Contact( "ENTRADAS Y SALIDAS"."BAJAR TAPA MANUAL"[1] )
   END_RUNG wire#w15
   RUNG wire#powerrail
      Contact( "HMI SALTAR PASO" )
   END_RUNG wire#w16
   RUNG wire#powerrail
      Contact( "HMI INICIAR CICLO PO" )
   END_RUNG wire#w17
   RUNG wire#powerrail
      Contact( "HMI INICIAR CICLO OP" )
   END_RUNG wire#w18
   RUNG wire#powerrail
      Contact( "HMI PAUSA" )
   END_RUNG wire#w19
   RUNG wire#powerrail
      Contact( "HMI CONTINUAR" )
   END_RUNG wire#w20
   RUNG wire#powerrail
      Contact( "HMI CANCELAR" )
   END_RUNG wire#w21
   RUNG wire#powerrail
      I_Contact( "PEMERG" )
   END_RUNG wire#w22
   RUNG wire#powerrail
      Contact( "HMI OK FIN DE CICLO" )
   END_RUNG wire#w23
   RUNG wire#powerrail
      Contact( "HMI OK CANCELAR" )
   END_RUNG wire#w24
   RUNG wire#powerrail
      Contact( "HMI RESET ACTUADORES MANUAL" )
   END_RUNG wire#w25
   RUNG wire#powerrail
      Contact(  )
   END_RUNG wire#w26
   RUNG wire#powerrail
      "ENVIO EQUIPO 1"(TEMPERATURAS := "ESTRUCTURAS Y ARREGLOS".TEMPERATURAS[1], ESTADO := "ESTRUCTURAS Y ARREGLOS".ESTADO[1]."COLOR EN HMI", "NIVEL AGUA" := "ESTRUCTURAS Y ARREGLOS".NIVEL[1], RECETA := "ESTRUCTURAS Y ARREGLOS"."CARGA RECETA"[1].NOMBRE, "NUM RECETA" := "ESTRUCTURAS Y ARREGLOS"."CARGA NUMERO RECETA"[1], "NUMERO EQUIPO" := 1, "ESTADO SERPENTINA" := "ESTADO".SALIDAS.COCINAS[1]."VAPOR SERPENTINA", "ESTADO VAPOR VIVO" := "ESTADO".SALIDAS.COCINAS[1]."VAPOR VIVO", TORRES := 1, PASOS := "ESTRUCTURAS Y ARREGLOS".ESTADO[1]."PASO ACTUAL", TIEMPO := "ESTRUCTURAS Y ARREGLOS".ESTADO[1]."TIEMPO TRANSCURRIDO", "T AGUA" => "COMUNICACION"."T AGUA", "T INGRESO" => "COMUNICACION"."T INGRESO", "T PRODUCTO" => "COMUNICACION"."T PROD", "ESTADO CICLO" => "COMUNICACION".ESTADO, NIVEL => "COMUNICACION".NIVEL, "NOMBRE RECETA" => "COMUNICACION"."NOMBRE RECETA", "NUMERO RECETA" => "COMUNICACION"."NUMERO RECETA", EQUIPO => "COMUNICACION"."NUMERO EQUIPO", SERPENTINA => "COMUNICACION".SERPENTINA, "VAPOR VIVO" => "COMUNICACION"."VAPOR VIVO", "NUMERO TORRES" => "COMUNICACION".TORRES, "CANTIDAD DE PASOS" => "COMUNICACION".PASOS, "TIEMPO TRANSCURRIDO" => "COMUNICACION"."TIEMPO TRANSCURRIDO")
   END_RUNG
   // the same network as SCL:
   // no checked SCL form for this network; see the picture
END_REGION

REGION Network 13: EQUIPO 2
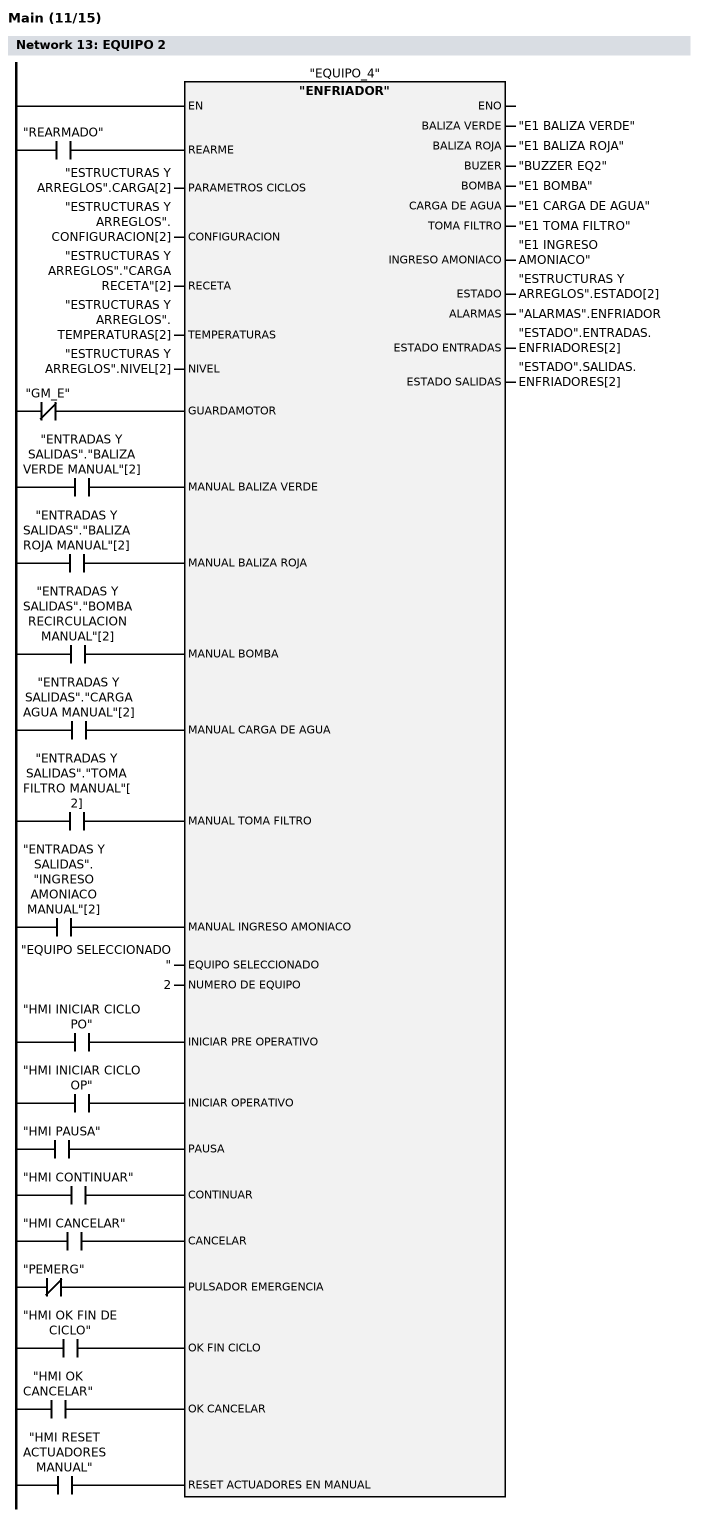
   RUNG wire#powerrail
      "EQUIPO_4"(REARME := wire#w1, GUARDAMOTOR := wire#w2, "MANUAL BALIZA VERDE" := wire#w3, "MANUAL BALIZA ROJA" := wire#w4, "MANUAL BOMBA" := wire#w5, "MANUAL CARGA DE AGUA" := wire#w6, "MANUAL TOMA FILTRO" := wire#w7, "MANUAL INGRESO AMONIACO" := wire#w8, "INICIAR PRE OPERATIVO" := wire#w9, "INICIAR OPERATIVO" := wire#w10, PAUSA := wire#w11, CONTINUAR := wire#w12, CANCELAR := wire#w13, "PULSADOR EMERGENCIA" := wire#w14, "OK FIN CICLO" := wire#w15, "OK CANCELAR" := wire#w16, "RESET ACTUADORES EN MANUAL" := wire#w17, "PARAMETROS CICLOS" := "ESTRUCTURAS Y ARREGLOS".CARGA[2], CONFIGURACION := "ESTRUCTURAS Y ARREGLOS".CONFIGURACION[2], RECETA := "ESTRUCTURAS Y ARREGLOS"."CARGA RECETA"[2], TEMPERATURAS := "ESTRUCTURAS Y ARREGLOS".TEMPERATURAS[2], NIVEL := "ESTRUCTURAS Y ARREGLOS".NIVEL[2], "EQUIPO SELECCIONADO" := "EQUIPO SELECCIONADO", "NUMERO DE EQUIPO" := 2, "BALIZA VERDE" => "E1 BALIZA VERDE", "BALIZA ROJA" => "E1 BALIZA ROJA", BUZER => "BUZZER EQ2", BOMBA => "E1 BOMBA", "CARGA DE AGUA" => "E1 CARGA DE AGUA", "TOMA FILTRO" => "E1 TOMA FILTRO", "INGRESO AMONIACO" => "E1 INGRESO AMONIACO", ESTADO => "ESTRUCTURAS Y ARREGLOS".ESTADO[2], ALARMAS => "ALARMAS".ENFRIADOR, "ESTADO ENTRADAS" => "ESTADO".ENTRADAS.ENFRIADORES[2], "ESTADO SALIDAS" => "ESTADO".SALIDAS.ENFRIADORES[2])
   END_RUNG
   RUNG wire#powerrail
      Contact( "REARMADO" )
   END_RUNG wire#w1
   RUNG wire#powerrail
      I_Contact( "GM_E" )
   END_RUNG wire#w2
   RUNG wire#powerrail
      Contact( "ENTRADAS Y SALIDAS"."BALIZA VERDE MANUAL"[2] )
   END_RUNG wire#w3
   RUNG wire#powerrail
      Contact( "ENTRADAS Y SALIDAS"."BALIZA ROJA MANUAL"[2] )
   END_RUNG wire#w4
   RUNG wire#powerrail
      Contact( "ENTRADAS Y SALIDAS"."BOMBA RECIRCULACION MANUAL"[2] )
   END_RUNG wire#w5
   RUNG wire#powerrail
      Contact( "ENTRADAS Y SALIDAS"."CARGA AGUA MANUAL"[2] )
   END_RUNG wire#w6
   RUNG wire#powerrail
      Contact( "ENTRADAS Y SALIDAS"."TOMA FILTRO MANUAL"[2] )
   END_RUNG wire#w7
   RUNG wire#powerrail
      Contact( "ENTRADAS Y SALIDAS"."INGRESO AMONIACO MANUAL"[2] )
   END_RUNG wire#w8
   RUNG wire#powerrail
      Contact( "HMI INICIAR CICLO PO" )
   END_RUNG wire#w9
   RUNG wire#powerrail
      Contact( "HMI INICIAR CICLO OP" )
   END_RUNG wire#w10
   RUNG wire#powerrail
      Contact( "HMI PAUSA" )
   END_RUNG wire#w11
   RUNG wire#powerrail
      Contact( "HMI CONTINUAR" )
   END_RUNG wire#w12
   RUNG wire#powerrail
      Contact( "HMI CANCELAR" )
   END_RUNG wire#w13
   RUNG wire#powerrail
      I_Contact( "PEMERG" )
   END_RUNG wire#w14
   RUNG wire#powerrail
      Contact( "HMI OK FIN DE CICLO" )
   END_RUNG wire#w15
   RUNG wire#powerrail
      Contact( "HMI OK CANCELAR" )
   END_RUNG wire#w16
   RUNG wire#powerrail
      Contact( "HMI RESET ACTUADORES MANUAL" )
   END_RUNG wire#w17
   // the same network as SCL:
   "EQUIPO_4"(REARME := "REARMADO",   // "ENFRIADOR"
              "PARAMETROS CICLOS" := "ESTRUCTURAS Y ARREGLOS".CARGA[2],
              CONFIGURACION := "ESTRUCTURAS Y ARREGLOS".CONFIGURACION[2],
              RECETA := "ESTRUCTURAS Y ARREGLOS"."CARGA RECETA"[2],
              TEMPERATURAS := "ESTRUCTURAS Y ARREGLOS".TEMPERATURAS[2],
              NIVEL := "ESTRUCTURAS Y ARREGLOS".NIVEL[2],
              GUARDAMOTOR := NOT "GM_E",
              "MANUAL BALIZA VERDE" := "ENTRADAS Y SALIDAS"."BALIZA VERDE MANUAL"[2],
              "MANUAL BALIZA ROJA" := "ENTRADAS Y SALIDAS"."BALIZA ROJA MANUAL"[2],
              "MANUAL BOMBA" := "ENTRADAS Y SALIDAS"."BOMBA RECIRCULACION MANUAL"[2],
              "MANUAL CARGA DE AGUA" := "ENTRADAS Y SALIDAS"."CARGA AGUA MANUAL"[2],
              "MANUAL TOMA FILTRO" := "ENTRADAS Y SALIDAS"."TOMA FILTRO MANUAL"[2],
              "MANUAL INGRESO AMONIACO" := "ENTRADAS Y SALIDAS"."INGRESO AMONIACO MANUAL"[2],
              "EQUIPO SELECCIONADO" := "EQUIPO SELECCIONADO",
              "NUMERO DE EQUIPO" := 2,
              "INICIAR PRE OPERATIVO" := "HMI INICIAR CICLO PO",
              "INICIAR OPERATIVO" := "HMI INICIAR CICLO OP",
              PAUSA := "HMI PAUSA",
              CONTINUAR := "HMI CONTINUAR",
              CANCELAR := "HMI CANCELAR",
              "PULSADOR EMERGENCIA" := NOT "PEMERG",
              "OK FIN CICLO" := "HMI OK FIN DE CICLO",
              "OK CANCELAR" := "HMI OK CANCELAR",
              "RESET ACTUADORES EN MANUAL" := "HMI RESET ACTUADORES MANUAL",
              "BALIZA VERDE" => "E1 BALIZA VERDE",
              "BALIZA ROJA" => "E1 BALIZA ROJA",
              BUZER => "BUZZER EQ2",
              BOMBA => "E1 BOMBA",
              "CARGA DE AGUA" => "E1 CARGA DE AGUA",
              "TOMA FILTRO" => "E1 TOMA FILTRO",
              "INGRESO AMONIACO" => "E1 INGRESO AMONIACO",
              ESTADO => "ESTRUCTURAS Y ARREGLOS".ESTADO[2],
              ALARMAS => "ALARMAS".ENFRIADOR,
              "ESTADO ENTRADAS" => "ESTADO".ENTRADAS.ENFRIADORES[2],
              "ESTADO SALIDAS" => "ESTADO".SALIDAS.ENFRIADORES[2]);
END_REGION

REGION Network 14: TRASPASO DE ESTADO DEL EQUIPO
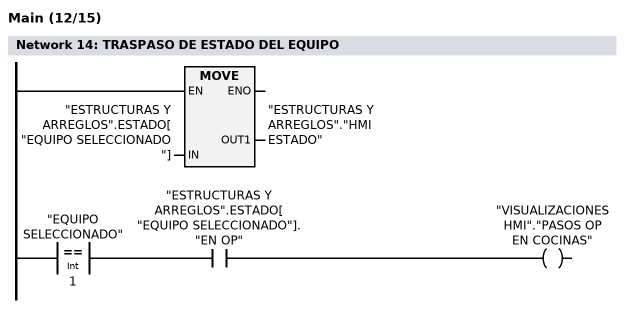
   RUNG wire#powerrail
      Move(in := "ESTRUCTURAS Y ARREGLOS".ESTADO["EQUIPO SELECCIONADO"], out1 => "ESTRUCTURAS Y ARREGLOS"."HMI ESTADO")
   END_RUNG
   RUNG wire#powerrail
      { S7_Templates := "SrcType := Int" } EQ_Contact(in1 := "EQUIPO SELECCIONADO", in2 := 1)
      Contact( "ESTRUCTURAS Y ARREGLOS".ESTADO["EQUIPO SELECCIONADO"]."EN OP" )
      Coil( "VISUALIZACIONES HMI"."PASOS OP EN COCINAS" )
   END_RUNG
   // the same network as SCL:
   "ESTRUCTURAS Y ARREGLOS"."HMI ESTADO" := "ESTRUCTURAS Y ARREGLOS".ESTADO["EQUIPO SELECCIONADO"];
   "VISUALIZACIONES HMI"."PASOS OP EN COCINAS" := ("EQUIPO SELECCIONADO" = 1) AND "ESTRUCTURAS Y ARREGLOS".ESTADO["EQUIPO SELECCIONADO"]."EN OP";
END_REGION

REGION Network 15: ACTIVACION DE SALIDAS DESDE HMI
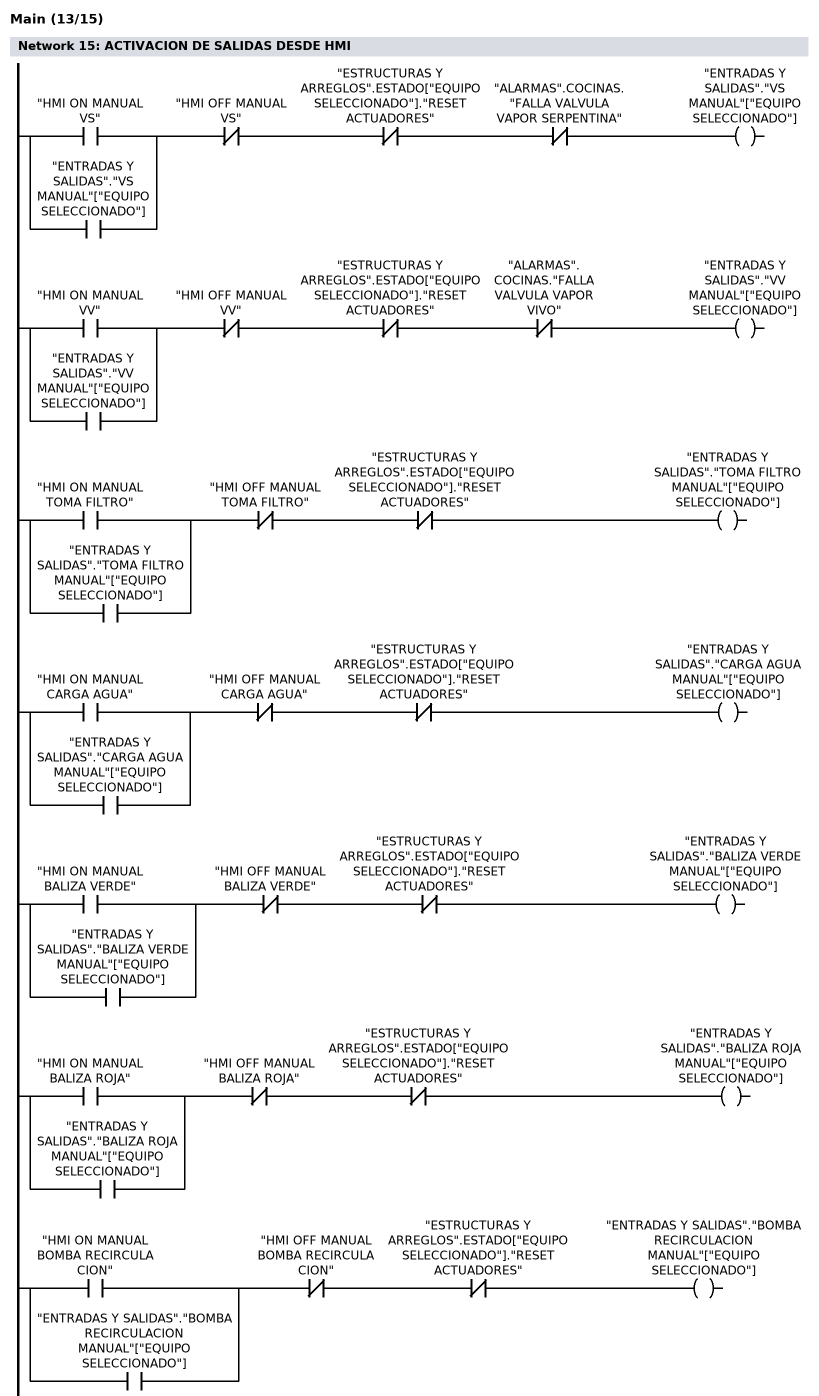
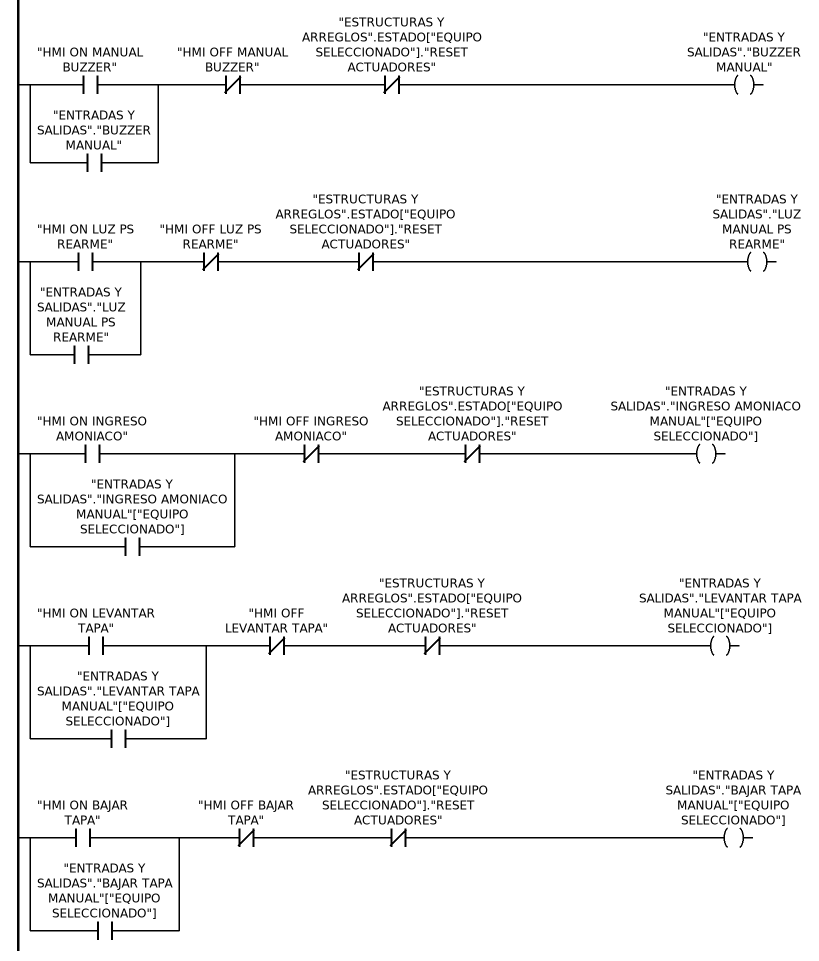
   RUNG wire#powerrail
      Contact( "HMI ON MANUAL VS" )
      wire#w1
      I_Contact( "HMI OFF MANUAL VS" )
      I_Contact( "ESTRUCTURAS Y ARREGLOS".ESTADO["EQUIPO SELECCIONADO"]."RESET ACTUADORES" )
      I_Contact( "ALARMAS".COCINAS."FALLA VALVULA VAPOR SERPENTINA" )
      Coil( "ENTRADAS Y SALIDAS"."VS MANUAL"["EQUIPO SELECCIONADO"] )
   END_RUNG
   RUNG wire#powerrail
      Contact( "ENTRADAS Y SALIDAS"."VS MANUAL"["EQUIPO SELECCIONADO"] )
   END_RUNG wire#w1
   RUNG wire#powerrail
      Contact( "HMI ON MANUAL VV" )
      wire#w2
      I_Contact( "HMI OFF MANUAL VV" )
      I_Contact( "ESTRUCTURAS Y ARREGLOS".ESTADO["EQUIPO SELECCIONADO"]."RESET ACTUADORES" )
      I_Contact( "ALARMAS".COCINAS."FALLA VALVULA VAPOR VIVO" )
      Coil( "ENTRADAS Y SALIDAS"."VV MANUAL"["EQUIPO SELECCIONADO"] )
   END_RUNG
   RUNG wire#powerrail
      Contact( "ENTRADAS Y SALIDAS"."VV MANUAL"["EQUIPO SELECCIONADO"] )
   END_RUNG wire#w2
   RUNG wire#powerrail
      Contact( "HMI ON MANUAL TOMA FILTRO" )
      wire#w3
      I_Contact( "HMI OFF MANUAL TOMA FILTRO" )
      I_Contact( "ESTRUCTURAS Y ARREGLOS".ESTADO["EQUIPO SELECCIONADO"]."RESET ACTUADORES" )
      Coil( "ENTRADAS Y SALIDAS"."TOMA FILTRO MANUAL"["EQUIPO SELECCIONADO"] )
   END_RUNG
   RUNG wire#powerrail
      Contact( "ENTRADAS Y SALIDAS"."TOMA FILTRO MANUAL"["EQUIPO SELECCIONADO"] )
   END_RUNG wire#w3
   RUNG wire#powerrail
      Contact( "HMI ON MANUAL CARGA AGUA" )
      wire#w4
      I_Contact( "HMI OFF MANUAL CARGA AGUA" )
      I_Contact( "ESTRUCTURAS Y ARREGLOS".ESTADO["EQUIPO SELECCIONADO"]."RESET ACTUADORES" )
      Coil( "ENTRADAS Y SALIDAS"."CARGA AGUA MANUAL"["EQUIPO SELECCIONADO"] )
   END_RUNG
   RUNG wire#powerrail
      Contact( "ENTRADAS Y SALIDAS"."CARGA AGUA MANUAL"["EQUIPO SELECCIONADO"] )
   END_RUNG wire#w4
   RUNG wire#powerrail
      Contact( "HMI ON MANUAL BALIZA VERDE" )
      wire#w5
      I_Contact( "HMI OFF MANUAL BALIZA VERDE" )
      I_Contact( "ESTRUCTURAS Y ARREGLOS".ESTADO["EQUIPO SELECCIONADO"]."RESET ACTUADORES" )
      Coil( "ENTRADAS Y SALIDAS"."BALIZA VERDE MANUAL"["EQUIPO SELECCIONADO"] )
   END_RUNG
   RUNG wire#powerrail
      Contact( "ENTRADAS Y SALIDAS"."BALIZA VERDE MANUAL"["EQUIPO SELECCIONADO"] )
   END_RUNG wire#w5
   RUNG wire#powerrail
      Contact( "HMI ON MANUAL BALIZA ROJA" )
      wire#w6
      I_Contact( "HMI OFF MANUAL BALIZA ROJA" )
      I_Contact( "ESTRUCTURAS Y ARREGLOS".ESTADO["EQUIPO SELECCIONADO"]."RESET ACTUADORES" )
      Coil( "ENTRADAS Y SALIDAS"."BALIZA ROJA MANUAL"["EQUIPO SELECCIONADO"] )
   END_RUNG
   RUNG wire#powerrail
      Contact( "ENTRADAS Y SALIDAS"."BALIZA ROJA MANUAL"["EQUIPO SELECCIONADO"] )
   END_RUNG wire#w6
   RUNG wire#powerrail
      Contact( "HMI ON MANUAL BOMBA RECIRCULACION" )
      wire#w7
      I_Contact( "HMI OFF MANUAL BOMBA RECIRCULACION" )
      I_Contact( "ESTRUCTURAS Y ARREGLOS".ESTADO["EQUIPO SELECCIONADO"]."RESET ACTUADORES" )
      Coil( "ENTRADAS Y SALIDAS"."BOMBA RECIRCULACION MANUAL"["EQUIPO SELECCIONADO"] )
   END_RUNG
   RUNG wire#powerrail
      Contact( "ENTRADAS Y SALIDAS"."BOMBA RECIRCULACION MANUAL"["EQUIPO SELECCIONADO"] )
   END_RUNG wire#w7
   RUNG wire#powerrail
      Contact( "HMI ON MANUAL BUZZER" )
      wire#w8
      I_Contact( "HMI OFF MANUAL BUZZER" )
      I_Contact( "ESTRUCTURAS Y ARREGLOS".ESTADO["EQUIPO SELECCIONADO"]."RESET ACTUADORES" )
      Coil( "ENTRADAS Y SALIDAS"."BUZZER MANUAL" )
   END_RUNG
   RUNG wire#powerrail
      Contact( "ENTRADAS Y SALIDAS"."BUZZER MANUAL" )
   END_RUNG wire#w8
   RUNG wire#powerrail
      Contact( "HMI ON LUZ PS REARME" )
      wire#w9
      I_Contact( "HMI OFF LUZ PS REARME" )
      I_Contact( "ESTRUCTURAS Y ARREGLOS".ESTADO["EQUIPO SELECCIONADO"]."RESET ACTUADORES" )
      Coil( "ENTRADAS Y SALIDAS"."LUZ MANUAL PS REARME" )
   END_RUNG
   RUNG wire#powerrail
      Contact( "ENTRADAS Y SALIDAS"."LUZ MANUAL PS REARME" )
   END_RUNG wire#w9
   RUNG wire#powerrail
      Contact( "HMI ON INGRESO AMONIACO" )
      wire#w10
      I_Contact( "HMI OFF INGRESO AMONIACO" )
      I_Contact( "ESTRUCTURAS Y ARREGLOS".ESTADO["EQUIPO SELECCIONADO"]."RESET ACTUADORES" )
      Coil( "ENTRADAS Y SALIDAS"."INGRESO AMONIACO MANUAL"["EQUIPO SELECCIONADO"] )
   END_RUNG
   RUNG wire#powerrail
      Contact( "ENTRADAS Y SALIDAS"."INGRESO AMONIACO MANUAL"["EQUIPO SELECCIONADO"] )
   END_RUNG wire#w10
   RUNG wire#powerrail
      Contact( "HMI ON LEVANTAR TAPA" )
      wire#w11
      I_Contact( "HMI OFF LEVANTAR TAPA" )
      I_Contact( "ESTRUCTURAS Y ARREGLOS".ESTADO["EQUIPO SELECCIONADO"]."RESET ACTUADORES" )
      Coil( "ENTRADAS Y SALIDAS"."LEVANTAR TAPA MANUAL"["EQUIPO SELECCIONADO"] )
   END_RUNG
   RUNG wire#powerrail
      Contact( "ENTRADAS Y SALIDAS"."LEVANTAR TAPA MANUAL"["EQUIPO SELECCIONADO"] )
   END_RUNG wire#w11
   RUNG wire#powerrail
      Contact( "HMI ON BAJAR TAPA" )
      wire#w12
      I_Contact( "HMI OFF BAJAR TAPA" )
      I_Contact( "ESTRUCTURAS Y ARREGLOS".ESTADO["EQUIPO SELECCIONADO"]."RESET ACTUADORES" )
      Coil( "ENTRADAS Y SALIDAS"."BAJAR TAPA MANUAL"["EQUIPO SELECCIONADO"] )
   END_RUNG
   RUNG wire#powerrail
      Contact( "ENTRADAS Y SALIDAS"."BAJAR TAPA MANUAL"["EQUIPO SELECCIONADO"] )
   END_RUNG wire#w12
   // the same network as SCL:
   "ENTRADAS Y SALIDAS"."VS MANUAL"["EQUIPO SELECCIONADO"] := ("HMI ON MANUAL VS" OR "ENTRADAS Y SALIDAS"."VS MANUAL"["EQUIPO SELECCIONADO"]) AND NOT "HMI OFF MANUAL VS" AND NOT "ESTRUCTURAS Y ARREGLOS".ESTADO["EQUIPO SELECCIONADO"]."RESET ACTUADORES" AND NOT "ALARMAS".COCINAS."FALLA VALVULA VAPOR SERPENTINA";
   "ENTRADAS Y SALIDAS"."VV MANUAL"["EQUIPO SELECCIONADO"] := ("HMI ON MANUAL VV" OR "ENTRADAS Y SALIDAS"."VV MANUAL"["EQUIPO SELECCIONADO"]) AND NOT "HMI OFF MANUAL VV" AND NOT "ESTRUCTURAS Y ARREGLOS".ESTADO["EQUIPO SELECCIONADO"]."RESET ACTUADORES" AND NOT "ALARMAS".COCINAS."FALLA VALVULA VAPOR VIVO";
   "ENTRADAS Y SALIDAS"."TOMA FILTRO MANUAL"["EQUIPO SELECCIONADO"] := ("HMI ON MANUAL TOMA FILTRO" OR "ENTRADAS Y SALIDAS"."TOMA FILTRO MANUAL"["EQUIPO SELECCIONADO"]) AND NOT "HMI OFF MANUAL TOMA FILTRO" AND NOT "ESTRUCTURAS Y ARREGLOS".ESTADO["EQUIPO SELECCIONADO"]."RESET ACTUADORES";
   "ENTRADAS Y SALIDAS"."CARGA AGUA MANUAL"["EQUIPO SELECCIONADO"] := ("HMI ON MANUAL CARGA AGUA" OR "ENTRADAS Y SALIDAS"."CARGA AGUA MANUAL"["EQUIPO SELECCIONADO"]) AND NOT "HMI OFF MANUAL CARGA AGUA" AND NOT "ESTRUCTURAS Y ARREGLOS".ESTADO["EQUIPO SELECCIONADO"]."RESET ACTUADORES";
   "ENTRADAS Y SALIDAS"."BALIZA VERDE MANUAL"["EQUIPO SELECCIONADO"] := ("HMI ON MANUAL BALIZA VERDE" OR "ENTRADAS Y SALIDAS"."BALIZA VERDE MANUAL"["EQUIPO SELECCIONADO"]) AND NOT "HMI OFF MANUAL BALIZA VERDE" AND NOT "ESTRUCTURAS Y ARREGLOS".ESTADO["EQUIPO SELECCIONADO"]."RESET ACTUADORES";
   "ENTRADAS Y SALIDAS"."BALIZA ROJA MANUAL"["EQUIPO SELECCIONADO"] := ("HMI ON MANUAL BALIZA ROJA" OR "ENTRADAS Y SALIDAS"."BALIZA ROJA MANUAL"["EQUIPO SELECCIONADO"]) AND NOT "HMI OFF MANUAL BALIZA ROJA" AND NOT "ESTRUCTURAS Y ARREGLOS".ESTADO["EQUIPO SELECCIONADO"]."RESET ACTUADORES";
   "ENTRADAS Y SALIDAS"."BOMBA RECIRCULACION MANUAL"["EQUIPO SELECCIONADO"] := ("HMI ON MANUAL BOMBA RECIRCULACION" OR "ENTRADAS Y SALIDAS"."BOMBA RECIRCULACION MANUAL"["EQUIPO SELECCIONADO"]) AND NOT "HMI OFF MANUAL BOMBA RECIRCULACION" AND NOT "ESTRUCTURAS Y ARREGLOS".ESTADO["EQUIPO SELECCIONADO"]."RESET ACTUADORES";
   "ENTRADAS Y SALIDAS"."BUZZER MANUAL" := ("HMI ON MANUAL BUZZER" OR "ENTRADAS Y SALIDAS"."BUZZER MANUAL") AND NOT "HMI OFF MANUAL BUZZER" AND NOT "ESTRUCTURAS Y ARREGLOS".ESTADO["EQUIPO SELECCIONADO"]."RESET ACTUADORES";
   "ENTRADAS Y SALIDAS"."LUZ MANUAL PS REARME" := ("HMI ON LUZ PS REARME" OR "ENTRADAS Y SALIDAS"."LUZ MANUAL PS REARME") AND NOT "HMI OFF LUZ PS REARME" AND NOT "ESTRUCTURAS Y ARREGLOS".ESTADO["EQUIPO SELECCIONADO"]."RESET ACTUADORES";
   "ENTRADAS Y SALIDAS"."INGRESO AMONIACO MANUAL"["EQUIPO SELECCIONADO"] := ("HMI ON INGRESO AMONIACO" OR "ENTRADAS Y SALIDAS"."INGRESO AMONIACO MANUAL"["EQUIPO SELECCIONADO"]) AND NOT "HMI OFF INGRESO AMONIACO" AND NOT "ESTRUCTURAS Y ARREGLOS".ESTADO["EQUIPO SELECCIONADO"]."RESET ACTUADORES";
   "ENTRADAS Y SALIDAS"."LEVANTAR TAPA MANUAL"["EQUIPO SELECCIONADO"] := ("HMI ON LEVANTAR TAPA" OR "ENTRADAS Y SALIDAS"."LEVANTAR TAPA MANUAL"["EQUIPO SELECCIONADO"]) AND NOT "HMI OFF LEVANTAR TAPA" AND NOT "ESTRUCTURAS Y ARREGLOS".ESTADO["EQUIPO SELECCIONADO"]."RESET ACTUADORES";
   "ENTRADAS Y SALIDAS"."BAJAR TAPA MANUAL"["EQUIPO SELECCIONADO"] := ("HMI ON BAJAR TAPA" OR "ENTRADAS Y SALIDAS"."BAJAR TAPA MANUAL"["EQUIPO SELECCIONADO"]) AND NOT "HMI OFF BAJAR TAPA" AND NOT "ESTRUCTURAS Y ARREGLOS".ESTADO["EQUIPO SELECCIONADO"]."RESET ACTUADORES";
END_REGION

REGION Network 16: ACTIVACION SALIDAS COMUNES A LOS EQUIPOS
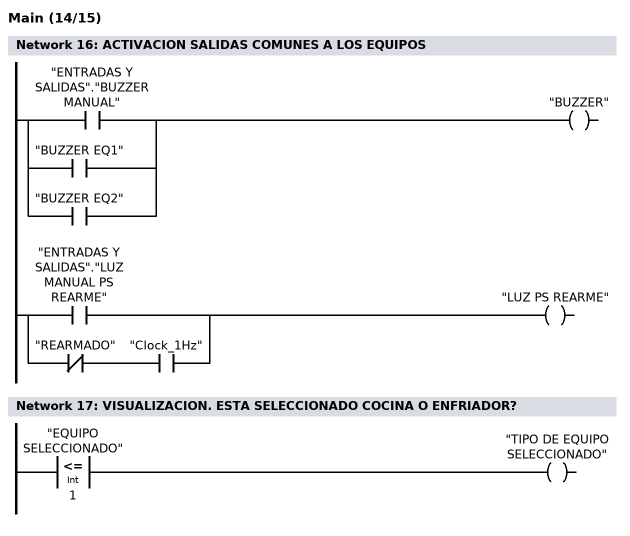
   RUNG wire#powerrail
      Contact( "ENTRADAS Y SALIDAS"."BUZZER MANUAL" )
      wire#w1
      Coil( "BUZZER" )
   END_RUNG
   RUNG wire#powerrail
      Contact( "BUZZER EQ1" )
   END_RUNG wire#w1
   RUNG wire#powerrail
      Contact( "BUZZER EQ2" )
   END_RUNG wire#w1
   RUNG wire#powerrail
      Contact( "ENTRADAS Y SALIDAS"."LUZ MANUAL PS REARME" )
      wire#w2
      Coil( "LUZ PS REARME" )
   END_RUNG
   RUNG wire#powerrail
      I_Contact( "REARMADO" )
      Contact( "Clock_1Hz" )
   END_RUNG wire#w2
   // the same network as SCL:
   "BUZZER" := "ENTRADAS Y SALIDAS"."BUZZER MANUAL" OR "BUZZER EQ1" OR "BUZZER EQ2";
   "LUZ PS REARME" := "ENTRADAS Y SALIDAS"."LUZ MANUAL PS REARME" OR (NOT "REARMADO" AND "Clock_1Hz");
END_REGION

REGION Network 17: VISUALIZACION. ESTA SELECCIONADO COCINA O ENFRIADOR?
   RUNG wire#powerrail
      { S7_Templates := "SrcType := Int" } LE_Contact(in1 := "EQUIPO SELECCIONADO", in2 := 1)
      Coil( "TIPO DE EQUIPO SELECCIONADO" )
   END_RUNG
   // the same network as SCL:
   "TIPO DE EQUIPO SELECCIONADO" := "EQUIPO SELECCIONADO" <= 1;
END_REGION

REGION Network 18: VISUALIZACIONES MODO MANUAL
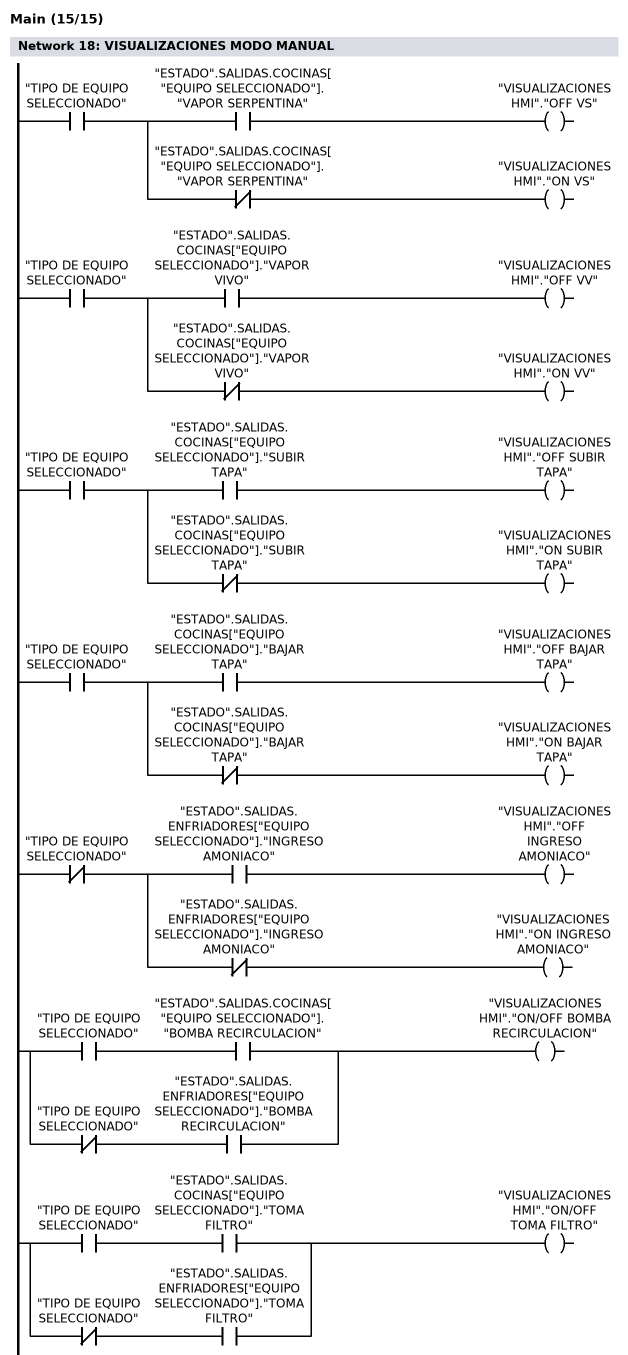
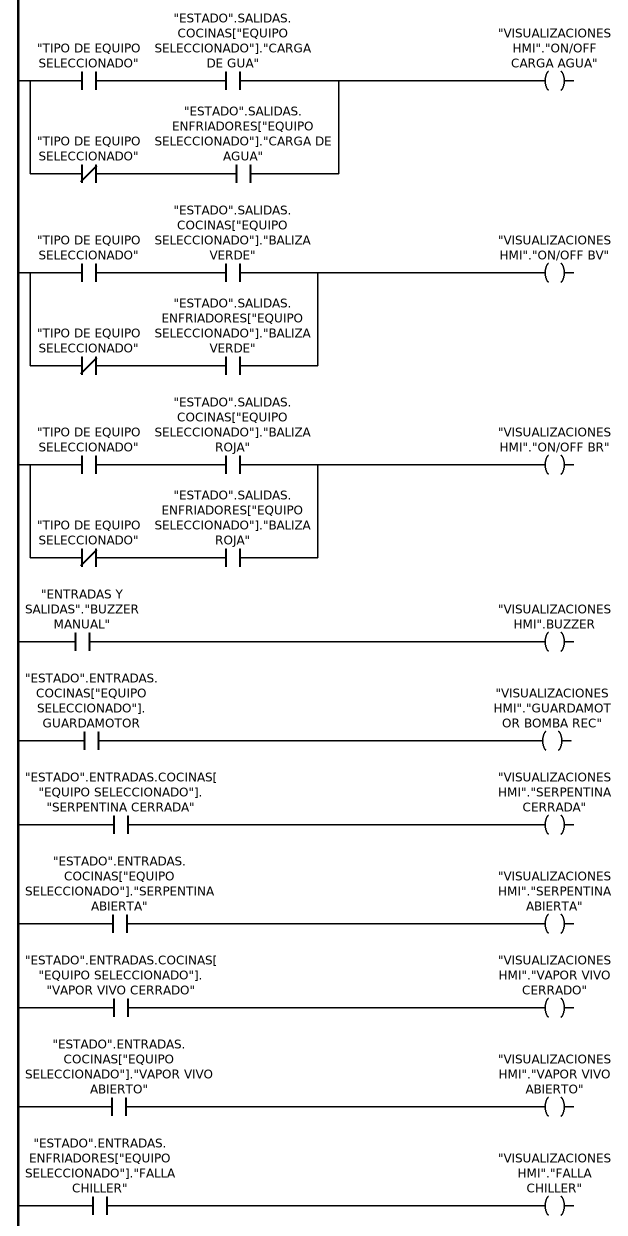
   RUNG wire#powerrail
      Contact( "TIPO DE EQUIPO SELECCIONADO" )
      wire#w1
      Contact( "ESTADO".SALIDAS.COCINAS["EQUIPO SELECCIONADO"]."VAPOR SERPENTINA" )
      Coil( "VISUALIZACIONES HMI"."OFF VS" )
   END_RUNG
   RUNG wire#w1
      I_Contact( "ESTADO".SALIDAS.COCINAS["EQUIPO SELECCIONADO"]."VAPOR SERPENTINA" )
      Coil( "VISUALIZACIONES HMI"."ON VS" )
   END_RUNG
   RUNG wire#powerrail
      Contact( "TIPO DE EQUIPO SELECCIONADO" )
      wire#w2
      Contact( "ESTADO".SALIDAS.COCINAS["EQUIPO SELECCIONADO"]."VAPOR VIVO" )
      Coil( "VISUALIZACIONES HMI"."OFF VV" )
   END_RUNG
   RUNG wire#w2
      I_Contact( "ESTADO".SALIDAS.COCINAS["EQUIPO SELECCIONADO"]."VAPOR VIVO" )
      Coil( "VISUALIZACIONES HMI"."ON VV" )
   END_RUNG
   RUNG wire#powerrail
      Contact( "TIPO DE EQUIPO SELECCIONADO" )
      wire#w3
      Contact( "ESTADO".SALIDAS.COCINAS["EQUIPO SELECCIONADO"]."SUBIR TAPA" )
      Coil( "VISUALIZACIONES HMI"."OFF SUBIR TAPA" )
   END_RUNG
   RUNG wire#w3
      I_Contact( "ESTADO".SALIDAS.COCINAS["EQUIPO SELECCIONADO"]."SUBIR TAPA" )
      Coil( "VISUALIZACIONES HMI"."ON SUBIR TAPA" )
   END_RUNG
   RUNG wire#powerrail
      Contact( "TIPO DE EQUIPO SELECCIONADO" )
      wire#w4
      Contact( "ESTADO".SALIDAS.COCINAS["EQUIPO SELECCIONADO"]."BAJAR TAPA" )
      Coil( "VISUALIZACIONES HMI"."OFF BAJAR TAPA" )
   END_RUNG
   RUNG wire#w4
      I_Contact( "ESTADO".SALIDAS.COCINAS["EQUIPO SELECCIONADO"]."BAJAR TAPA" )
      Coil( "VISUALIZACIONES HMI"."ON BAJAR TAPA" )
   END_RUNG
   RUNG wire#powerrail
      I_Contact( "TIPO DE EQUIPO SELECCIONADO" )
      wire#w5
      Contact( "ESTADO".SALIDAS.ENFRIADORES["EQUIPO SELECCIONADO"]."INGRESO AMONIACO" )
      Coil( "VISUALIZACIONES HMI"."OFF INGRESO AMONIACO" )
   END_RUNG
   RUNG wire#w5
      I_Contact( "ESTADO".SALIDAS.ENFRIADORES["EQUIPO SELECCIONADO"]."INGRESO AMONIACO" )
      Coil( "VISUALIZACIONES HMI"."ON INGRESO AMONIACO" )
   END_RUNG
   RUNG wire#powerrail
      Contact( "TIPO DE EQUIPO SELECCIONADO" )
      Contact( "ESTADO".SALIDAS.COCINAS["EQUIPO SELECCIONADO"]."BOMBA RECIRCULACION" )
      wire#w6
      Coil( "VISUALIZACIONES HMI"."ON/OFF BOMBA RECIRCULACION" )
   END_RUNG
   RUNG wire#powerrail
      I_Contact( "TIPO DE EQUIPO SELECCIONADO" )
      Contact( "ESTADO".SALIDAS.ENFRIADORES["EQUIPO SELECCIONADO"]."BOMBA RECIRCULACION" )
   END_RUNG wire#w6
   RUNG wire#powerrail
      Contact( "TIPO DE EQUIPO SELECCIONADO" )
      Contact( "ESTADO".SALIDAS.COCINAS["EQUIPO SELECCIONADO"]."TOMA FILTRO" )
      wire#w7
      Coil( "VISUALIZACIONES HMI"."ON/OFF TOMA FILTRO" )
   END_RUNG
   RUNG wire#powerrail
      I_Contact( "TIPO DE EQUIPO SELECCIONADO" )
      Contact( "ESTADO".SALIDAS.ENFRIADORES["EQUIPO SELECCIONADO"]."TOMA FILTRO" )
   END_RUNG wire#w7
   RUNG wire#powerrail
      Contact( "TIPO DE EQUIPO SELECCIONADO" )
      Contact( "ESTADO".SALIDAS.COCINAS["EQUIPO SELECCIONADO"]."CARGA DE GUA" )
      wire#w8
      Coil( "VISUALIZACIONES HMI"."ON/OFF CARGA AGUA" )
   END_RUNG
   RUNG wire#powerrail
      I_Contact( "TIPO DE EQUIPO SELECCIONADO" )
      Contact( "ESTADO".SALIDAS.ENFRIADORES["EQUIPO SELECCIONADO"]."CARGA DE AGUA" )
   END_RUNG wire#w8
   RUNG wire#powerrail
      Contact( "TIPO DE EQUIPO SELECCIONADO" )
      Contact( "ESTADO".SALIDAS.COCINAS["EQUIPO SELECCIONADO"]."BALIZA VERDE" )
      wire#w9
      Coil( "VISUALIZACIONES HMI"."ON/OFF BV" )
   END_RUNG
   RUNG wire#powerrail
      I_Contact( "TIPO DE EQUIPO SELECCIONADO" )
      Contact( "ESTADO".SALIDAS.ENFRIADORES["EQUIPO SELECCIONADO"]."BALIZA VERDE" )
   END_RUNG wire#w9
   RUNG wire#powerrail
      Contact( "TIPO DE EQUIPO SELECCIONADO" )
      Contact( "ESTADO".SALIDAS.COCINAS["EQUIPO SELECCIONADO"]."BALIZA ROJA" )
      wire#w10
      Coil( "VISUALIZACIONES HMI"."ON/OFF BR" )
   END_RUNG
   RUNG wire#powerrail
      I_Contact( "TIPO DE EQUIPO SELECCIONADO" )
      Contact( "ESTADO".SALIDAS.ENFRIADORES["EQUIPO SELECCIONADO"]."BALIZA ROJA" )
   END_RUNG wire#w10
   RUNG wire#powerrail
      Contact( "ENTRADAS Y SALIDAS"."BUZZER MANUAL" )
      Coil( "VISUALIZACIONES HMI".BUZZER )
   END_RUNG
   RUNG wire#powerrail
      Contact( "ESTADO".ENTRADAS.COCINAS["EQUIPO SELECCIONADO"].GUARDAMOTOR )
      Coil( "VISUALIZACIONES HMI"."GUARDAMOTOR BOMBA REC" )
   END_RUNG
   RUNG wire#powerrail
      Contact( "ESTADO".ENTRADAS.COCINAS["EQUIPO SELECCIONADO"]."SERPENTINA CERRADA" )
      Coil( "VISUALIZACIONES HMI"."SERPENTINA CERRADA" )
   END_RUNG
   RUNG wire#powerrail
      Contact( "ESTADO".ENTRADAS.COCINAS["EQUIPO SELECCIONADO"]."SERPENTINA ABIERTA" )
      Coil( "VISUALIZACIONES HMI"."SERPENTINA ABIERTA" )
   END_RUNG
   RUNG wire#powerrail
      Contact( "ESTADO".ENTRADAS.COCINAS["EQUIPO SELECCIONADO"]."VAPOR VIVO CERRADO" )
      Coil( "VISUALIZACIONES HMI"."VAPOR VIVO CERRADO" )
   END_RUNG
   RUNG wire#powerrail
      Contact( "ESTADO".ENTRADAS.COCINAS["EQUIPO SELECCIONADO"]."VAPOR VIVO ABIERTO" )
      Coil( "VISUALIZACIONES HMI"."VAPOR VIVO ABIERTO" )
   END_RUNG
   RUNG wire#powerrail
      Contact( "ESTADO".ENTRADAS.ENFRIADORES["EQUIPO SELECCIONADO"]."FALLA CHILLER" )
      Coil( "VISUALIZACIONES HMI"."FALLA CHILLER" )
   END_RUNG
   // the same network as SCL:
   "VISUALIZACIONES HMI"."OFF VS" := "TIPO DE EQUIPO SELECCIONADO" AND "ESTADO".SALIDAS.COCINAS["EQUIPO SELECCIONADO"]."VAPOR SERPENTINA";
   "VISUALIZACIONES HMI"."ON VS" := "TIPO DE EQUIPO SELECCIONADO" AND NOT "ESTADO".SALIDAS.COCINAS["EQUIPO SELECCIONADO"]."VAPOR SERPENTINA";
   "VISUALIZACIONES HMI"."OFF VV" := "TIPO DE EQUIPO SELECCIONADO" AND "ESTADO".SALIDAS.COCINAS["EQUIPO SELECCIONADO"]."VAPOR VIVO";
   "VISUALIZACIONES HMI"."ON VV" := "TIPO DE EQUIPO SELECCIONADO" AND NOT "ESTADO".SALIDAS.COCINAS["EQUIPO SELECCIONADO"]."VAPOR VIVO";
   "VISUALIZACIONES HMI"."OFF SUBIR TAPA" := "TIPO DE EQUIPO SELECCIONADO" AND "ESTADO".SALIDAS.COCINAS["EQUIPO SELECCIONADO"]."SUBIR TAPA";
   "VISUALIZACIONES HMI"."ON SUBIR TAPA" := "TIPO DE EQUIPO SELECCIONADO" AND NOT "ESTADO".SALIDAS.COCINAS["EQUIPO SELECCIONADO"]."SUBIR TAPA";
   "VISUALIZACIONES HMI"."OFF BAJAR TAPA" := "TIPO DE EQUIPO SELECCIONADO" AND "ESTADO".SALIDAS.COCINAS["EQUIPO SELECCIONADO"]."BAJAR TAPA";
   "VISUALIZACIONES HMI"."ON BAJAR TAPA" := "TIPO DE EQUIPO SELECCIONADO" AND NOT "ESTADO".SALIDAS.COCINAS["EQUIPO SELECCIONADO"]."BAJAR TAPA";
   #_w1 := NOT "TIPO DE EQUIPO SELECCIONADO";
   "VISUALIZACIONES HMI"."OFF INGRESO AMONIACO" := #_w1 AND "ESTADO".SALIDAS.ENFRIADORES["EQUIPO SELECCIONADO"]."INGRESO AMONIACO";
   "VISUALIZACIONES HMI"."ON INGRESO AMONIACO" := #_w1 AND NOT "ESTADO".SALIDAS.ENFRIADORES["EQUIPO SELECCIONADO"]."INGRESO AMONIACO";
   "VISUALIZACIONES HMI"."ON/OFF BOMBA RECIRCULACION" := ("TIPO DE EQUIPO SELECCIONADO" AND "ESTADO".SALIDAS.COCINAS["EQUIPO SELECCIONADO"]."BOMBA RECIRCULACION") OR (NOT "TIPO DE EQUIPO SELECCIONADO" AND "ESTADO".SALIDAS.ENFRIADORES["EQUIPO SELECCIONADO"]."BOMBA RECIRCULACION");
   "VISUALIZACIONES HMI"."ON/OFF TOMA FILTRO" := ("TIPO DE EQUIPO SELECCIONADO" AND "ESTADO".SALIDAS.COCINAS["EQUIPO SELECCIONADO"]."TOMA FILTRO") OR (NOT "TIPO DE EQUIPO SELECCIONADO" AND "ESTADO".SALIDAS.ENFRIADORES["EQUIPO SELECCIONADO"]."TOMA FILTRO");
   "VISUALIZACIONES HMI"."ON/OFF CARGA AGUA" := ("TIPO DE EQUIPO SELECCIONADO" AND "ESTADO".SALIDAS.COCINAS["EQUIPO SELECCIONADO"]."CARGA DE GUA") OR (NOT "TIPO DE EQUIPO SELECCIONADO" AND "ESTADO".SALIDAS.ENFRIADORES["EQUIPO SELECCIONADO"]."CARGA DE AGUA");
   "VISUALIZACIONES HMI"."ON/OFF BV" := ("TIPO DE EQUIPO SELECCIONADO" AND "ESTADO".SALIDAS.COCINAS["EQUIPO SELECCIONADO"]."BALIZA VERDE") OR (NOT "TIPO DE EQUIPO SELECCIONADO" AND "ESTADO".SALIDAS.ENFRIADORES["EQUIPO SELECCIONADO"]."BALIZA VERDE");
   "VISUALIZACIONES HMI"."ON/OFF BR" := ("TIPO DE EQUIPO SELECCIONADO" AND "ESTADO".SALIDAS.COCINAS["EQUIPO SELECCIONADO"]."BALIZA ROJA") OR (NOT "TIPO DE EQUIPO SELECCIONADO" AND "ESTADO".SALIDAS.ENFRIADORES["EQUIPO SELECCIONADO"]."BALIZA ROJA");
   "VISUALIZACIONES HMI".BUZZER := "ENTRADAS Y SALIDAS"."BUZZER MANUAL";
   "VISUALIZACIONES HMI"."GUARDAMOTOR BOMBA REC" := "ESTADO".ENTRADAS.COCINAS["EQUIPO SELECCIONADO"].GUARDAMOTOR;
   "VISUALIZACIONES HMI"."SERPENTINA CERRADA" := "ESTADO".ENTRADAS.COCINAS["EQUIPO SELECCIONADO"]."SERPENTINA CERRADA";
   "VISUALIZACIONES HMI"."SERPENTINA ABIERTA" := "ESTADO".ENTRADAS.COCINAS["EQUIPO SELECCIONADO"]."SERPENTINA ABIERTA";
   "VISUALIZACIONES HMI"."VAPOR VIVO CERRADO" := "ESTADO".ENTRADAS.COCINAS["EQUIPO SELECCIONADO"]."VAPOR VIVO CERRADO";
   "VISUALIZACIONES HMI"."VAPOR VIVO ABIERTO" := "ESTADO".ENTRADAS.COCINAS["EQUIPO SELECCIONADO"]."VAPOR VIVO ABIERTO";
   "VISUALIZACIONES HMI"."FALLA CHILLER" := "ESTADO".ENTRADAS.ENFRIADORES["EQUIPO SELECCIONADO"]."FALLA CHILLER";
END_REGION
END_ORGANIZATION_BLOCK

(* ===== HMI "HMI_RT_1" =====
system functions are stored by id; their names below are inferred from use
connection "HMI_Connection_1": ETHERNET, SMART_S7_1200_OMS

HMI tags "Default tag table"
   "INICIAR CICLO" : Bool = PLC "HMI INICIAR CICLO PO" AT %M300.0, 1 s
   "VISUALIZACIONES HMI_ON/OFF CARGA AGUA" : Bool = PLC "VISUALIZACIONES HMI"."ON/OFF CARGA AGUA", 1 s
   "VISUALIZACIONES HMI_ON/OFF BR" : Bool = PLC "VISUALIZACIONES HMI"."ON/OFF BR", 1 s
   "VISUALIZACIONES HMI_ON/OFF BV" : Bool = PLC "VISUALIZACIONES HMI"."ON/OFF BV", 1 s
   "VISUALIZACIONES HMI_ON/OFF TOMA FILTRO" : Bool = PLC "VISUALIZACIONES HMI"."ON/OFF TOMA FILTRO", 1 s
   "VISUALIZACIONES HMI_BUZZER" : Bool = PLC "VISUALIZACIONES HMI".BUZZER, 1 s
   "HMI ON MANUAL VS" : Bool = PLC "HMI ON MANUAL VS" AT %M300.4, 1 s
   "HMI ON MANUAL VV" : Bool = PLC "HMI ON MANUAL VV" AT %M300.5, 1 s
   "HMI ON MANUAL CARGA AGUA" : Bool = PLC "HMI ON MANUAL CARGA AGUA" AT %M300.6, 1 s
   "HMI ON MANUAL BALIZA ROJA" : Bool = PLC "HMI ON MANUAL BALIZA ROJA" AT %M301.1, 1 s
   "HMI ON MANUAL BALIZA VERDE" : Bool = PLC "HMI ON MANUAL BALIZA VERDE" AT %M301.0, 1 s
   "HMI ON MANUAL TOMA FILTRO" : Bool = PLC "HMI ON MANUAL TOMA FILTRO" AT %M300.7, 1 s
   "HMI ON MANUAL BUZZER" : Bool = PLC "HMI ON MANUAL BUZZER" AT %M301.2, 1 s
   "HMI OFF MANUAL VS" : Bool = PLC "HMI OFF MANUAL VS" AT %M301.3, 1 s
   "HMI OFF MANUAL VV" : Bool = PLC "HMI OFF MANUAL VV" AT %M301.4, 1 s
   "HMI OFF MANUAL CARGA AGUA" : Bool = PLC "HMI OFF MANUAL CARGA AGUA" AT %M301.5, 1 s
   "HMI OFF MANUAL BALIZA ROJA" : Bool = PLC "HMI OFF MANUAL BALIZA ROJA" AT %M302.0, 1 s
   "HMI OFF MANUAL BALIZA VERDE" : Bool = PLC "HMI OFF MANUAL BALIZA VERDE" AT %M301.7, 1 s
   "HMI OFF MANUAL TOMA FILTRO" : Bool = PLC "HMI OFF MANUAL TOMA FILTRO" AT %M301.6, 1 s
   "HMI OFF BUZZER" : Bool = PLC "HMI OFF BUZZER" AT %M304.4, 1 s
   "EQUIPO MANUAL" : Int = PLC "EQUIPO MANUAL" AT %MW710, 1 s
   "HMI SIGUIENTE EQUIPO MM" : Bool = PLC "HMI SIGUIENTE EQUIPO MM" AT %M302.2, 1 s
   "HMI ANTERIOR EQUIPO MM" : Bool = PLC "HMI ANTERIOR EQUIPO MM" AT %M302.3, 1 s
   "HMI AUMENTAR EQUIPO" : Bool = PLC "HMI AUMENTAR EQUIPO" AT %M305.0, 1 s
   "HMI DISMINUIR EQUIPO" : Bool = PLC "HMI DISMINUIR EQUIPO" AT %M305.1, 1 s
   "EQUIPO SELECCIONADO" : Int = PLC "EQUIPO SELECCIONADO" AT %MW700, 1 s
   "HMI SEL ANT RECETA" : Bool = PLC "HMI SEL ANT RECETA" AT %M304.1, 1 s
   "HMI SEL SIG RECETA" : Bool = PLC "HMI SEL SIG RECETA" AT %M304.0, 1 s
   "HMI RECETA SELECCIONADA" : Int = PLC "HMI RECETA SELECCIONADA" AT %MW746, 1 s
   "HMI RECETA ANTERIOR" : Bool = PLC "HMI RECETA ANTERIOR" AT %M305.3, 1 s
   "HMI RECETA SIGUIENTE" : Bool = PLC "HMI RECETA SIGUIENTE" AT %M305.2, 1 s
   "HMI NUMERO RECETA" : Int = PLC "HMI NUMERO RECETA" AT %MW742, 1 s
   "HMI RESTAR PASO" : Bool = PLC "HMI RESTAR PASO" AT %M305.6, 1 s
   "HMI SUMAR PASO" : Bool = PLC "HMI SUMAR PASO" AT %M305.5, 1 s
   "ESTRUCTURAS Y ARREGLOS_HMI EDICION RECETAS_PASOS" : Int = PLC "ESTRUCTURAS Y ARREGLOS"."HMI EDICION RECETAS".PASOS, 1 s
   "ESTRUCTURAS Y ARREGLOS_HMI EDICION RECETAS_NOMBRE" : String[254] = PLC "ESTRUCTURAS Y ARREGLOS"."HMI EDICION RECETAS".NOMBRE, 1 s
   "ESTRUCTURAS Y ARREGLOS_HMI EDICION RECETAS_TEMP AGUA{1}" : Int = PLC "ESTRUCTURAS Y ARREGLOS"."HMI EDICION RECETAS"."TEMP AGUA"[1], 1 s
   "ESTRUCTURAS Y ARREGLOS_HMI EDICION RECETAS_TEMP AGUA{2}" : Int = PLC "ESTRUCTURAS Y ARREGLOS"."HMI EDICION RECETAS"."TEMP AGUA"[2], 1 s
   "ESTRUCTURAS Y ARREGLOS_HMI EDICION RECETAS_TEMP AGUA{3}" : Int = PLC "ESTRUCTURAS Y ARREGLOS"."HMI EDICION RECETAS"."TEMP AGUA"[3], 1 s
   "ESTRUCTURAS Y ARREGLOS_HMI EDICION RECETAS_TEMP AGUA{4}" : Int = PLC "ESTRUCTURAS Y ARREGLOS"."HMI EDICION RECETAS"."TEMP AGUA"[4], 1 s
   "ESTRUCTURAS Y ARREGLOS_HMI EDICION RECETAS_TIEMPO CORTE{1}" : Int = PLC "ESTRUCTURAS Y ARREGLOS"."HMI EDICION RECETAS"."TIEMPO CORTE"[1], 1 s
   "ESTRUCTURAS Y ARREGLOS_HMI EDICION RECETAS_TIEMPO CORTE{2}" : Int = PLC "ESTRUCTURAS Y ARREGLOS"."HMI EDICION RECETAS"."TIEMPO CORTE"[2], 1 s
   "ESTRUCTURAS Y ARREGLOS_HMI EDICION RECETAS_TIEMPO CORTE{3}" : Int = PLC "ESTRUCTURAS Y ARREGLOS"."HMI EDICION RECETAS"."TIEMPO CORTE"[3], 1 s
   "ESTRUCTURAS Y ARREGLOS_HMI EDICION RECETAS_TIEMPO CORTE{4}" : Int = PLC "ESTRUCTURAS Y ARREGLOS"."HMI EDICION RECETAS"."TIEMPO CORTE"[4], 1 s
   "ESTRUCTURAS Y ARREGLOS_HMI EDICION RECETAS_TEMP PRODUCTO{1}" : Int = PLC "ESTRUCTURAS Y ARREGLOS"."HMI EDICION RECETAS"."TEMP PRODUCTO"[1], 1 s
   "ESTRUCTURAS Y ARREGLOS_HMI EDICION RECETAS_TEMP PRODUCTO{2}" : Int = PLC "ESTRUCTURAS Y ARREGLOS"."HMI EDICION RECETAS"."TEMP PRODUCTO"[2], 1 s
   "ESTRUCTURAS Y ARREGLOS_HMI EDICION RECETAS_TEMP PRODUCTO{3}" : Int = PLC "ESTRUCTURAS Y ARREGLOS"."HMI EDICION RECETAS"."TEMP PRODUCTO"[3], 1 s
   "ESTRUCTURAS Y ARREGLOS_HMI EDICION RECETAS_TEMP PRODUCTO{4}" : Int = PLC "ESTRUCTURAS Y ARREGLOS"."HMI EDICION RECETAS"."TEMP PRODUCTO"[4], 1 s
   "ESTRUCTURAS Y ARREGLOS_HMI EDICION RECETAS_TIPO CORTE{1}" : Bool = PLC "ESTRUCTURAS Y ARREGLOS"."HMI EDICION RECETAS"."TIPO CORTE"[1], 1 s
   "ESTRUCTURAS Y ARREGLOS_HMI EDICION RECETAS_TIPO CORTE{2}" : Bool = PLC "ESTRUCTURAS Y ARREGLOS"."HMI EDICION RECETAS"."TIPO CORTE"[2], 1 s
   "ESTRUCTURAS Y ARREGLOS_HMI EDICION RECETAS_TIPO CORTE{3}" : Bool = PLC "ESTRUCTURAS Y ARREGLOS"."HMI EDICION RECETAS"."TIPO CORTE"[3], 1 s
   "ESTRUCTURAS Y ARREGLOS_HMI EDICION RECETAS_TIPO CORTE{4}" : Bool = PLC "ESTRUCTURAS Y ARREGLOS"."HMI EDICION RECETAS"."TIPO CORTE"[4], 1 s
   "ESTRUCTURAS Y ARREGLOS_HMI CARGA_TEMPERATURAS_TEMPERATURA AGUA SC" : Real = PLC "ESTRUCTURAS Y ARREGLOS"."HMI CARGA".TEMPERATURAS."TEMPERATURA AGUA SC", 1 s
   "ESTRUCTURAS Y ARREGLOS_HMI CARGA_TEMPERATURAS_TEMPERATURA INGRESO SC" : Real = PLC "ESTRUCTURAS Y ARREGLOS"."HMI CARGA".TEMPERATURAS."TEMPERATURA INGRESO SC", 1 s
   "ESTRUCTURAS Y ARREGLOS_HMI CARGA_TEMPERATURAS_TEMPERATURA PRODUCTO SC" : Real = PLC "ESTRUCTURAS Y ARREGLOS"."HMI CARGA".TEMPERATURAS."TEMPERATURA PRODUCTO SC", 1 s
   "ESTRUCTURAS Y ARREGLOS_CORRECCIONES{1}_TEMPERATURA AGUA" : Real = PLC "ESTRUCTURAS Y ARREGLOS".CORRECCIONES[1]."TEMPERATURA AGUA", 1 s
   "ESTRUCTURAS Y ARREGLOS_HMI CARGA_TEMPERATURAS_TEMPERATURA AGUA" : Real = PLC "ESTRUCTURAS Y ARREGLOS"."HMI CARGA".TEMPERATURAS."TEMPERATURA AGUA", 1 s
   "ESTRUCTURAS Y ARREGLOS_HMI CARGA_TEMPERATURAS_TEMPERATURA INGRESO" : Real = PLC "ESTRUCTURAS Y ARREGLOS"."HMI CARGA".TEMPERATURAS."TEMPERATURA INGRESO", 1 s
   "ESTRUCTURAS Y ARREGLOS_HMI CARGA_TEMPERATURAS_TEMPERATURA PRODUCTO" : Real = PLC "ESTRUCTURAS Y ARREGLOS"."HMI CARGA".TEMPERATURAS."TEMPERATURA PRODUCTO", 1 s
   "ESTRUCTURAS Y ARREGLOS_CORRECCIONES HMI_TEMPERATURA AGUA SC" : Real = PLC "ESTRUCTURAS Y ARREGLOS"."CORRECCIONES HMI"."TEMPERATURA AGUA SC", 1 s
   "ESTRUCTURAS Y ARREGLOS_CORRECCIONES HMI_TEMPERATURA INGRESO SC" : Real = PLC "ESTRUCTURAS Y ARREGLOS"."CORRECCIONES HMI"."TEMPERATURA INGRESO SC", 1 s
   "ESTRUCTURAS Y ARREGLOS_CORRECCIONES HMI_TEMPERATURA PRODUCTO SC" : Real = PLC "ESTRUCTURAS Y ARREGLOS"."CORRECCIONES HMI"."TEMPERATURA PRODUCTO SC", 1 s
   "ESTRUCTURAS Y ARREGLOS_HMI CONFIGURACION_NIVEL OP" : Int = PLC "ESTRUCTURAS Y ARREGLOS"."HMI CONFIGURACION"."NIVEL OP", 1 s
   "ESTRUCTURAS Y ARREGLOS_HMI CONFIGURACION_VENTANA" : Int = PLC "ESTRUCTURAS Y ARREGLOS"."HMI CONFIGURACION".VENTANA, 1 s
   "ESTRUCTURAS Y ARREGLOS_HMI CONFIGURACION_NIVEL PO{1}" : Int = PLC "ESTRUCTURAS Y ARREGLOS"."HMI CONFIGURACION"."NIVEL PO"[1], 1 s
   "ESTRUCTURAS Y ARREGLOS_HMI CONFIGURACION_NIVEL PO{2}" : Int = PLC "ESTRUCTURAS Y ARREGLOS"."HMI CONFIGURACION"."NIVEL PO"[2], 1 s
   "ESTRUCTURAS Y ARREGLOS_HMI CONFIGURACION_NIVEL PO{3}" : Int = PLC "ESTRUCTURAS Y ARREGLOS"."HMI CONFIGURACION"."NIVEL PO"[3], 1 s
   "ESTRUCTURAS Y ARREGLOS_TEMPERATURAS{1}_TEMPERATURA AGUA" : Real = PLC "ESTRUCTURAS Y ARREGLOS".TEMPERATURAS[1]."TEMPERATURA AGUA", 1 s
   "ESTRUCTURAS Y ARREGLOS_TEMPERATURAS{1}_TEMPERATURA INGRESO" : Real = PLC "ESTRUCTURAS Y ARREGLOS".TEMPERATURAS[1]."TEMPERATURA INGRESO", 1 s
   "ESTRUCTURAS Y ARREGLOS_TEMPERATURAS{1}_TEMPERATURA PRODUCTO" : Real = PLC "ESTRUCTURAS Y ARREGLOS".TEMPERATURAS[1]."TEMPERATURA PRODUCTO", 1 s
   "ESTRUCTURAS Y ARREGLOS_TEMPERATURAS{2}_TEMPERATURA AGUA" : Real = PLC "ESTRUCTURAS Y ARREGLOS".TEMPERATURAS[2]."TEMPERATURA AGUA", 1 s
   "ESTRUCTURAS Y ARREGLOS_TEMPERATURAS{2}_TEMPERATURA INGRESO" : Real = PLC "ESTRUCTURAS Y ARREGLOS".TEMPERATURAS[2]."TEMPERATURA INGRESO", 1 s
   "ESTRUCTURAS Y ARREGLOS_TEMPERATURAS{2}_TEMPERATURA PRODUCTO" : Real = PLC "ESTRUCTURAS Y ARREGLOS".TEMPERATURAS[2]."TEMPERATURA PRODUCTO", 1 s
   "HMI VER EQUIPO 1" : Bool = PLC "HMI VER EQUIPO 1" AT %M303.1, 1 s
   "HMI VER EQUIPO 2" : Bool = PLC "HMI VER EQUIPO 2" AT %M303.2, 1 s
   "HMI VER EQUIPO 3" : Bool = PLC "HMI VER EQUIPO 3" AT %M303.3, 1 s
   "HMI VER EQUIPO 4" : Bool = PLC "HMI VER EQUIPO 4" AT %M303.4, 1 s
   "ESTRUCTURAS Y ARREGLOS_CARGA RECETA{1}_NOMBRE" : String[254] = PLC "ESTRUCTURAS Y ARREGLOS"."CARGA RECETA"[1].NOMBRE, 1 s
   "ESTRUCTURAS Y ARREGLOS_CARGA RECETA{2}_NOMBRE" : String[254] = PLC "ESTRUCTURAS Y ARREGLOS"."CARGA RECETA"[2].NOMBRE, 1 s
   "ESTRUCTURAS Y ARREGLOS_CARGA{1}_CANTIDAD DE TORRES" : Int = PLC "ESTRUCTURAS Y ARREGLOS".CARGA[1]."CANTIDAD DE TORRES", 1 s
   "ESTRUCTURAS Y ARREGLOS_CARGA{2}_CANTIDAD DE TORRES" : Int = PLC "ESTRUCTURAS Y ARREGLOS".CARGA[2]."CANTIDAD DE TORRES", 1 s
   "CALIBRACION SN MAXIMO" : Bool = PLC "CALIBRACION SN MAXIMO" AT %M304.5, 1 s
   "CALIBRACION SN MINIMO" : Bool = PLC "CALIBRACION SN MINIMO" AT %M304.6, 1 s
   "HMI NIVEL" : Int = PLC "HMI NIVEL" AT %MW748, 1 s
   "VISUALIZACIONES HMI_GUARDAMOTOR" : Bool = PLC "VISUALIZACIONES HMI"."GUARDAMOTOR BOMBA REC", 1 s
   "VISUALIZACIONES HMI_SERPENTINA ABIERTA" : Bool = PLC "VISUALIZACIONES HMI"."SERPENTINA ABIERTA", 1 s
   "VISUALIZACIONES HMI_SERPENTINA CERRADA" : Bool = PLC "VISUALIZACIONES HMI"."SERPENTINA CERRADA", 1 s
   "VISUALIZACIONES HMI_VAPOR VIVO ABIERTO" : Bool = PLC "VISUALIZACIONES HMI"."VAPOR VIVO ABIERTO", 1 s
   "VISUALIZACIONES HMI_VAPOR VIVO CERRADO" : Bool = PLC "VISUALIZACIONES HMI"."VAPOR VIVO CERRADO", 1 s
   "PRARM" : Bool = PLC PRARM AT %I1.0, 1 s
   "PEMERG" : Bool = PLC PEMERG AT %I1.2, 1 s
   "HMI ON LUZ PS REARME" : Bool = PLC "HMI ON LUZ PS REARME" AT %M305.7, 1 s
   "HMI OFF LUZ PS REARME" : Bool = PLC "HMI OFF LUZ PS REARME" AT %M306.1, 1 s
   "HMI ON LUZ REARME" : Bool = PLC "HMI ON LUZ REARME" AT %M1501.0, 1 s
   "ENTRADAS Y SALIDAS_LUZ MANUAL PS REARME" : Bool = PLC "ENTRADAS Y SALIDAS"."LUZ MANUAL PS REARME", 1 s
   "HMI OFF MANUAL BUZZER" : Bool = PLC "HMI OFF MANUAL BUZZER" AT %M302.1, 1 s
   "ESTRUCTURAS Y ARREGLOS_NIVEL{1}" : Int = PLC "ESTRUCTURAS Y ARREGLOS".NIVEL[1], 1 s
   "ESTRUCTURAS Y ARREGLOS_NIVEL{2}" : Int = PLC "ESTRUCTURAS Y ARREGLOS".NIVEL[2], 1 s
   "TIPO DE EQUIPO SELECCIONADO" : Bool = PLC "TIPO DE EQUIPO SELECCIONADO" AT %M307.2, 1 s
   "VISUALIZACIONES HMI_ON VS" : Bool = PLC "VISUALIZACIONES HMI"."ON VS", 1 s
   "VISUALIZACIONES HMI_ON VV" : Bool = PLC "VISUALIZACIONES HMI"."ON VV", 1 s
   "VISUALIZACIONES HMI_ON BOMBA RECIRCULACION" : Bool = PLC "VISUALIZACIONES HMI"."ON/OFF BOMBA RECIRCULACION", 1 s
   "VISUALIZACIONES HMI_OFF VS" : Bool = PLC "VISUALIZACIONES HMI"."OFF VS", 1 s
   "VISUALIZACIONES HMI_OFF VV" : Bool = PLC "VISUALIZACIONES HMI"."OFF VV", 1 s
   "HMI ON MANUAL BI" : Bool = PLC "HMI ON MANUAL BI" AT %M306.6, 1 s
   "HMI ON MANUAL BE" : Bool = PLC "HMI ON MANUAL BE" AT %M307.0, 1 s
   "HMI ON MANUAL V INGRESO" : Bool = PLC "HMI ON MANUAL V INGRESO" AT %M306.4, 1 s
   "VISUALIZACIONES HMI_ON BOMBA INGRESO" : Bool = PLC "VISUALIZACIONES HMI"."ON BOMBA INGRESO", 1 s
   "VISUALIZACIONES HMI_ON BOMBA EGRESO" : Bool = PLC "VISUALIZACIONES HMI"."ON BOMBA EGRESO", 1 s
   "VISUALIZACIONES HMI_ON V INGRESO" : Bool = PLC "VISUALIZACIONES HMI"."ON V INGRESO", 1 s
   "VISUALIZACIONES HMI_ON V EGRESO" : Bool = PLC "VISUALIZACIONES HMI"."ON V EGRESO", 1 s
   "VISUALIZACIONES HMI_OFF BOMBA INGRESO" : Bool = PLC "VISUALIZACIONES HMI"."OFF BOMBA INGRESO", 1 s
   "VISUALIZACIONES HMI_OFF BOMBA EGRESO" : Bool = PLC "VISUALIZACIONES HMI"."OFF BOMBA EGRESO", 1 s
   "VISUALIZACIONES HMI_OFF V EGRESO" : Bool = PLC "VISUALIZACIONES HMI"."OFF V EGRESO", 1 s
   "VISUALIZACIONES HMI_OFF V INGRESO" : Bool = PLC "VISUALIZACIONES HMI"."OFF V INGRESO", 1 s
   "HMI OFF MANUAL BI" : Bool = PLC "HMI OFF MANUAL BI" AT %M306.7, 1 s
   "HMI OFF MANUAL BE" : Bool = PLC "HMI OFF MANUAL BE" AT %M307.1, 1 s
   "HMI OFF MANUAL V INGRESO" : Bool = PLC "HMI OFF MANUAL V INGRESO" AT %M306.5, 1 s
   "ESTRUCTURAS Y ARREGLOS_HMI CONFIGURACION_DELAY" : Int = PLC "ESTRUCTURAS Y ARREGLOS"."HMI CONFIGURACION".DELAY, 1 s
   "ESTRUCTURAS Y ARREGLOS_HMI CONFIGURACION_HISTERESIS" : DInt = PLC "ESTRUCTURAS Y ARREGLOS"."HMI CONFIGURACION".HISTERESIS, 1 s
   "ESTRUCTURAS Y ARREGLOS_HMI CONFIGURACION_TIEMPO MAXIMO CICLO" : Int = PLC "ESTRUCTURAS Y ARREGLOS"."HMI CONFIGURACION"."TIEMPO MAXIMO CICLO", 1 s
   "ESTRUCTURAS Y ARREGLOS_HMI CONFIGURACION_NIVEL CRITICO" : Int = PLC "ESTRUCTURAS Y ARREGLOS"."HMI CONFIGURACION"."NIVEL CRITICO PO", 1 s
   "HMI AUMENTAR CANT TORRES" : Bool = PLC "HMI AUMENTAR CANT TORRES" AT %M303.6, 1 s
   "DISMINUIR CANT TORRES" : Bool = PLC "HMI DISMINUIR CANT TORRES" AT %M303.7, 1 s
   "ESTRUCTURAS Y ARREGLOS_HMI EDICION RECETAS_TIEMPO CORTE ENFRIADO" : Int = PLC "ESTRUCTURAS Y ARREGLOS"."HMI EDICION RECETAS"."TIEMPO CORTE ENFRIADO", 1 s
   "ESTRUCTURAS Y ARREGLOS_HMI EDICION RECETAS_TEMP CORTE ENFRIADO" : Int = PLC "ESTRUCTURAS Y ARREGLOS"."HMI EDICION RECETAS"."TEMP CORTE ENFRIADO", 1 s
   "ESTRUCTURAS Y ARREGLOS_HMI CARGA_NIVEL MINIMO" : Int = PLC "ESTRUCTURAS Y ARREGLOS"."HMI CARGA"."NIVEL MINIMO", 1 s
   "ESTRUCTURAS Y ARREGLOS_HMI CARGA RECETA_NOMBRE" : String[254] = PLC "ESTRUCTURAS Y ARREGLOS"."HMI MOSTRAR RECETA".NOMBRE, 1 s
   "ESTRUCTURAS Y ARREGLOS_HMI CARGA_NOMBRE RECETA" : String[254] = PLC "ESTRUCTURAS Y ARREGLOS"."HMI CARGA"."NOMBRE RECETA", 1 s
   "ESTRUCTURAS Y ARREGLOS_HMI CARGA_CANTIDAD DE TORRES" : Int = PLC "ESTRUCTURAS Y ARREGLOS"."HMI CARGA"."CANTIDAD DE TORRES", 1 s
   "HMI PAUSA" : Bool = PLC "HMI PAUSA" AT %M302.6, 1 s
   "ESTRUCTURAS Y ARREGLOS_HMI CARGA_TIPO DE CORTE" : Bool = PLC "ESTRUCTURAS Y ARREGLOS"."HMI CARGA"."TIPO DE CORTE", 1 s
   "ESTRUCTURAS Y ARREGLOS_HMI EDICION RECETAS_TIPO CORTE ENFRIADO" : Bool = PLC "ESTRUCTURAS Y ARREGLOS"."HMI EDICION RECETAS"."TIPO CORTE ENFRIADO", 1 s
   "VISUALIZACIONES HMI_1 PASO RECETA" : Bool = PLC "VISUALIZACIONES HMI"."1 PASO RECETA", 1 s
   "VISUALIZACIONES HMI_2 PASOS RECETA" : Bool = PLC "VISUALIZACIONES HMI"."2 PASOS RECETA", 1 s
   "VISUALIZACIONES HMI_3 PASOS RECETA" : Bool = PLC "VISUALIZACIONES HMI"."3 PASOS RECETA", 1 s
   "VISUALIZACIONES HMI_4 PASOS RECETA" : Bool = PLC "VISUALIZACIONES HMI"."4 PASOS RECETA", 1 s
   "VISUALIZACIONES HMI_TIPO DE CORTE PASO 1" : Bool = PLC "VISUALIZACIONES HMI"."CORTE TEMP PASO 1", 1 s
   "VISUALIZACIONES HMI_TIPO DE CORTE PASO 2" : Bool = PLC "VISUALIZACIONES HMI"."CORTE TEMP PASO 2", 1 s
   "VISUALIZACIONES HMI_TIPO DE CORTE PASO 3" : Bool = PLC "VISUALIZACIONES HMI"."CORTE TEMP PASO 3", 1 s
   "VISUALIZACIONES HMI_TIPO DE CORTE PASO 4" : Bool = PLC "VISUALIZACIONES HMI"."CORTE TEMP PASO 4", 1 s
   "VISUALIZACIONES HMI_CORTE TIEMPO PASO 1" : Bool = PLC "VISUALIZACIONES HMI"."CORTE TIEMPO PASO 1", 1 s
   "VISUALIZACIONES HMI_CORTE TIEMPO PASO 2" : Bool = PLC "VISUALIZACIONES HMI"."CORTE TIEMPO PASO 2", 1 s
   "VISUALIZACIONES HMI_CORTE TIEMPO PASO 3" : Bool = PLC "VISUALIZACIONES HMI"."CORTE TIEMPO PASO 3", 1 s
   "VISUALIZACIONES HMI_CORTE TIEMPO PASO 4" : Bool = PLC "VISUALIZACIONES HMI"."CORTE TIEMPO PASO 4", 1 s
   "VISUALIZACIONES HMI_CORTE TIEMPO ENFRIADOR" : Bool = PLC "VISUALIZACIONES HMI"."CORTE TIEMPO ENFRIADOR", 1 s
   "VISUALIZACIONES HMI_CORTE TEMP ENFRIADOR" : Bool = PLC "VISUALIZACIONES HMI"."CORTE TEMP ENFRIADOR", 1 s
   "ESTRUCTURAS Y ARREGLOS_HMI CARGA_TEMPERATURA CORTE PC" : Int = PLC "ESTRUCTURAS Y ARREGLOS"."HMI CARGA"."TEMPERATURA CORTE PC", 1 s
   "ESTRUCTURAS Y ARREGLOS_HMI CARGA_TIEMPO CORTE PC" : Int = PLC "ESTRUCTURAS Y ARREGLOS"."HMI CARGA"."TIEMPO CORTE PC", 1 s
   "HMI CONTINUAR" : Bool = PLC "HMI CONTINUAR" AT %M302.7, 1 s
   "HMI CANCELAR" : Bool = PLC "HMI CANCELAR" AT %M303.0, 1 s
   "HMI INICIAR CICLO OP" : Bool = PLC "HMI INICIAR CICLO OP" AT %M300.3, 1 s
   "ESTRUCTURAS Y ARREGLOS_HMI ESTADO_TIEMPO TRANSCURRIDO" : DInt = PLC "ESTRUCTURAS Y ARREGLOS"."HMI ESTADO"."TIEMPO TRANSCURRIDO", 1 s
   "ESTRUCTURAS Y ARREGLOS_ESTADO{1}_EQUIPO" : String[254] = PLC "ESTRUCTURAS Y ARREGLOS".ESTADO[1].EQUIPO, 1 s
   "ESTRUCTURAS Y ARREGLOS_ESTADO{2}_EQUIPO" : String[254] = PLC "ESTRUCTURAS Y ARREGLOS".ESTADO[2].EQUIPO, 1 s
   "ESTRUCTURAS Y ARREGLOS_ESTADO{1}_TIEMPO TRANSCURRIDO" : DInt = PLC "ESTRUCTURAS Y ARREGLOS".ESTADO[1]."TIEMPO TRANSCURRIDO", 1 s
   "ESTRUCTURAS Y ARREGLOS_ESTADO{2}_TIEMPO TRANSCURRIDO" : DInt = PLC "ESTRUCTURAS Y ARREGLOS".ESTADO[2]."TIEMPO TRANSCURRIDO", 1 s
   "ESTRUCTURAS Y ARREGLOS_HMI ESTADO_EN CICLO" : Bool = PLC "ESTRUCTURAS Y ARREGLOS"."HMI ESTADO"."EN CICLO", 1 s
   "ESTRUCTURAS Y ARREGLOS_HMI ESTADO_EQUIPO" : String[254] = PLC "ESTRUCTURAS Y ARREGLOS"."HMI ESTADO".EQUIPO, 1 s
   "ESTRUCTURAS Y ARREGLOS_HMI ESTADO_TIPO DE CORTE" : String[254] = PLC "ESTRUCTURAS Y ARREGLOS"."HMI ESTADO"."TIPO DE CORTE", 1 s
   "ESTRUCTURAS Y ARREGLOS_HMI ESTADO_EN PO" : Bool = PLC "ESTRUCTURAS Y ARREGLOS"."HMI ESTADO"."EN PO", 1 s
   "ESTRUCTURAS Y ARREGLOS_HMI ESTADO_EN OP" : Bool = PLC "ESTRUCTURAS Y ARREGLOS"."HMI ESTADO"."EN OP", 1 s
   "ESTRUCTURAS Y ARREGLOS_HMI ESTADO_PULSADOR PAUSA" : Bool = PLC "ESTRUCTURAS Y ARREGLOS"."HMI ESTADO"."PULSADOR PAUSA", 1 s
   "ESTRUCTURAS Y ARREGLOS_HMI ESTADO_PULSADOR CONTINUAR" : Bool = PLC "ESTRUCTURAS Y ARREGLOS"."HMI ESTADO"."PULSADOR CONTINUAR", 1 s
   "ESTRUCTURAS Y ARREGLOS_HMI ESTADO_PULSADOR CANCELAR" : Bool = PLC "ESTRUCTURAS Y ARREGLOS"."HMI ESTADO"."PULSADOR CANCELAR", 1 s
   "VISUALIZACIONES HMI_PASOS OP EN COCINAS" : Bool = PLC "VISUALIZACIONES HMI"."PASOS OP EN COCINAS", 1 s
   "ESTRUCTURAS Y ARREGLOS_HMI ESTADO_CICLO FINALIZADO" : Bool = PLC "ESTRUCTURAS Y ARREGLOS"."HMI ESTADO"."CICLO FINALIZADO", 1 s
   "HMI OK CANCELAR" : Bool = PLC "HMI OK CANCELAR" AT %M307.4, 1 s
   "ESTRUCTURAS Y ARREGLOS_HMI ESTADO_CICLO CANCELADO" : Bool = PLC "ESTRUCTURAS Y ARREGLOS"."HMI ESTADO"."CICLO CANCELADO", 1 s
   "HMI OK FIN DE CICLO" : Bool = PLC "HMI OK FIN DE CICLO" AT %M307.3, 1 s
   "ESTRUCTURAS Y ARREGLOS_HMI NOMBRE EQUIPO" : String[254] = PLC "ESTRUCTURAS Y ARREGLOS"."HMI NOMBRE EQUIPO", 1 s
   "ESTRUCTURAS Y ARREGLOS_HMI ESTADO_MANUAL ACTIVO" : Bool = PLC "ESTRUCTURAS Y ARREGLOS"."HMI ESTADO"."MANUAL ACTIVO", 1 s
   "HMI RESET ACTUADORES MANUAL" : Bool = PLC "HMI RESET ACTUADORES MANUAL" AT %M307.6, 1 s
   "HMI SALTAR PASO" : Bool = PLC "HMI SALTAR PASO" AT %M307.7, 1 s
   "VISUALIZACIONES HMI_GRAFICOS" : Int = PLC "VISUALIZACIONES HMI".GRAFICOS, 1 s
   "ESTRUCTURAS Y ARREGLOS_HMI ESTADO_PASO ACTUAL" : Int = PLC "ESTRUCTURAS Y ARREGLOS"."HMI ESTADO"."PASO ACTUAL", 1 s
   "VISUALIZACIONES HMI_LIM INF CANT TORRES" : Bool = PLC "VISUALIZACIONES HMI"."LIM INF CANT TORRES", 1 s
   "VISUALIZACIONES HMI_LIM SUP CANT TORRES" : Bool = PLC "VISUALIZACIONES HMI"."LIM SUP CANT TORRES", 1 s
   "VISUALIZACIONES HMI_LIM INF EQUIPO SEL" : Bool = PLC "VISUALIZACIONES HMI"."LIM INF EQUIPO SEL", 1 s
   "VISUALIZACIONES HMI_LIM SUP EQUIPO SEL" : Bool = PLC "VISUALIZACIONES HMI"."LIM SUP EQUIPO SEL", 1 s
   "HMI VISUALIZAR RECETA" : Bool = PLC "HMI VISUALIZAR RECETA" AT %M1701.0, 1 s
   "VISUALIZACIONES HMI_ANTERIOR RECETA" : Bool = PLC "VISUALIZACIONES HMI"."ANTERIOR RECETA", 1 s
   "VISUALIZACIONES HMI_SIGUIENTE RECETA" : Bool = PLC "VISUALIZACIONES HMI"."SIGUIENTE RECETA", 1 s
   "VISUALIZACIONES HMI_ANTERIOR PASO" : Bool = PLC "VISUALIZACIONES HMI"."ANTERIOR PASO", 1 s
   "VISUALIZACIONES HMI_SIGUIENTE PASO" : Bool = PLC "VISUALIZACIONES HMI"."SIGUIENTE PASO", 1 s
   "VISUALIZACIONES HMI_BLOQUEO EDICION RECETAS" : Bool = PLC "VISUALIZACIONES HMI"."BLOQUEO EDICION RECETAS", 1 s
   "HMI VOLVER" : Bool = PLC "HMI VOLVER" AT %M1701.2, 1 s
   "HMI RECETARIO" : Bool = PLC "HMI RECETARIO" AT %M1701.1, 1 s
   "ESTRUCTURAS Y ARREGLOS_ESTADO{1}_COLOR EN HMI" : Int = PLC "ESTRUCTURAS Y ARREGLOS".ESTADO[1]."COLOR EN HMI", 1 s
   "ESTRUCTURAS Y ARREGLOS_ESTADO{2}_COLOR EN HMI" : Int = PLC "ESTRUCTURAS Y ARREGLOS".ESTADO[2]."COLOR EN HMI", 1 s
   "ESTRUCTURAS Y ARREGLOS_HMI CARGA_VAPOR VIVO" : Bool = PLC "ESTRUCTURAS Y ARREGLOS"."HMI CARGA"."VAPOR VIVO", 1 s
   "ESTRUCTURAS Y ARREGLOS_HMI CONFIGURACION_NIVEL CRITICO OP" : Int = PLC "ESTRUCTURAS Y ARREGLOS"."HMI CONFIGURACION"."NIVEL CRITICO OP", 1 s
   "PANTALLA BLOQUEO" : Int = PLC "IMAGEN BLOQUEO" AT %MW770, 1 s
      on ChangeValue: ActivateScreenByNumber("PANTALLA BLOQUEO", 1)
   "DIAS RESTANTES" : DInt = PLC "DIAS RESTANTES" AT %MD762, 1 s
   "HMI CONTRASEÑA INGRESADA" : DInt = PLC "HMI CONTRASEÑA INGRESADA" AT %MD758, 1 s
   "VISUALIZACIONES HMI_OFF SUBIR TAPA" : Bool = PLC "VISUALIZACIONES HMI"."OFF SUBIR TAPA", 1 s
   "VISUALIZACIONES HMI_ON BAJAR TAPA" : Bool = PLC "VISUALIZACIONES HMI"."ON BAJAR TAPA", 1 s
   "VISUALIZACIONES HMI_ON SUBIR TAPA" : Bool = PLC "VISUALIZACIONES HMI"."ON SUBIR TAPA", 1 s
   "VISUALIZACIONES HMI_OFF BAJAR TAPA" : Bool = PLC "VISUALIZACIONES HMI"."OFF BAJAR TAPA", 1 s
   "HMI ON MANUAL BOMBA RECIRCULACION" : Bool = PLC "HMI ON MANUAL BOMBA RECIRCULACION" AT %M302.4, 1 s
   "HMI OFF MANUAL BOMBA RECIRCULACION" : Bool = PLC "HMI OFF MANUAL BOMBA RECIRCULACION" AT %M302.5, 1 s
   "HMI ON INGRESO AMONIACO" : Bool = PLC "HMI ON INGRESO AMONIACO" AT %M306.2, 1 s
   "HMI OFF INGRESO AMONIACO" : Bool = PLC "HMI OFF INGRESO AMONIACO" AT %M306.3, 1 s
   "VISUALIZACIONES HMI_OFF INGRESO AMONIACO" : Bool = PLC "VISUALIZACIONES HMI"."OFF INGRESO AMONIACO", 1 s
   "VISUALIZACIONES HMI_ON INGRESO AMONIACO" : Bool = PLC "VISUALIZACIONES HMI"."ON INGRESO AMONIACO", 1 s
   "HMI ON LEVANTAR TAPA" : Bool = PLC "HMI ON LEVANTAR TAPA" AT %M1701.3, 1 s
   "HMI OFF LEVANTAR TAPA" : Bool = PLC "HMI OFF LEVANTAR TAPA" AT %M1701.4, 1 s
   "HMI ON BAJAR TAPA" : Bool = PLC "HMI ON BAJAR TAPA" AT %M1701.5, 1 s
   "HMI OFF BAJAR TAPA" : Bool = PLC "HMI OFF BAJAR TAPA" AT %M1701.6, 1 s

HMI tags "ALARMAS"
   "ALARMAS_EQ1" : UInt AT %DB5.DBW0, 1 s
   "ALARMAS_EQ2" : UInt AT %DB5.DBW2, 1 s
   "ALARMAS GENERAL" : UInt AT %DB5.DBW4, 1 s

discrete alarms
   10: 'Parada de emergencia activa. Desactivela para habilitar el rearmado', class Errors, trigger "ALARMAS GENERAL" bit 8
   20: 'Presionar pulsador de rearme', class Errors, trigger "ALARMAS GENERAL" bit 9
   2: 'Se detecto una falla en la apertura/cierre de la valvula de vapor de serpentina de la cocina 1. Revise su estado', class Errors, trigger "ALARMAS_EQ1" bit 8
   3: 'Se detecto una falla en la apertura/cierre de la valvula de vapor vivo de la cocina 1. Revise su estado', class Errors, trigger "ALARMAS_EQ1" bit 9
   11: 'Falla en la bomba de recirculacion de la cocina 1. Revisar Guardamotor', class Errors, trigger "ALARMAS_EQ1" bit 10
   13: 'Nivel critico de agua e insuficiente para continuar el ciclo en cocina 1. Puede haberse generado alguna perdida', class Errors, trigger "ALARMAS_EQ1" bit 11
   15: 'Falla en la bomba de recirculacion del enfriador 1. Revisar Guardamotor', class Errors, trigger "ALARMAS_EQ2" bit 8
   24: 'Nivel critico de agua e insuficiente para continuar el ciclo en enfriador 1. Puede haberse generado alguna perdida', class Errors, trigger "ALARMAS_EQ2" bit 10
   26: 'Se detecto una falla en el sensor de temperatura de agua en la cocina 1. Verifique su estado', class Errors, trigger "ALARMAS_EQ1" bit 12
   27: 'Se detecto una falla en el sensor de temperatura de ingreso en la cocina 1. Verifique su estado', class Errors, trigger "ALARMAS_EQ1" bit 13
   28: 'Se detecto una falla en el sensor de temperatura de producto en la cocina 1. Verifique su estado', class Errors, trigger "ALARMAS_EQ1" bit 14
   32: 'Se detecto una falla en el sensor de temperatura de agua en el enfriador 1. Verifique su estado', class Errors, trigger "ALARMAS_EQ2" bit 11
   33: 'Se detecto una falla en el sensor de temperatura de ingreso en el enfriador 1. Verifique su estado', class Errors, trigger "ALARMAS_EQ2" bit 12
   34: 'Se detecto una falla en el sensor de temperatura de producto en el enfriador 1. Verifique su estado', class Errors, trigger "ALARMAS_EQ2" bit 13
   40: 'El sistema no detecto una carga de agua en la cocina 1. Por favor cancele el ciclo , vuelva a comenzar y verifique la entrada de agua', class Errors, trigger "ALARMAS_EQ1" bit 15
   42: 'El sistema no detecto una carga de agua en el enfriador 1. Por favor cancele el ciclo , vuelva a comenzar y verifique la entrada de agua', class Errors, trigger "ALARMAS_EQ2" bit 14

text list "list_TIPOCORTE": 0 'TEMPERATURA'; 1 'TIEMPO'

screen "MANUAL" 800x480, template "Template_1"
   TextField "Text field_1" at 449,406 size 161x22; Text 'VAPOR SERPENTINA'
      Visibility <- "TIPO DE EQUIPO SELECCIONADO"
   TextField "Text field_2" at 509,445 size 101x22; Text 'VAPOR VIVO'
      Visibility <- "TIPO DE EQUIPO SELECCIONADO"
   TextField "Text field_23" at 500,367 size 110x22; Text 'CERRAR TAPA'
      Visibility <- "TIPO DE EQUIPO SELECCIONADO"
   TextField "Text field_20" at 482,328 size 128x22; Text 'LEVANTAR TAPA'
      Visibility <- "TIPO DE EQUIPO SELECCIONADO"
   TextField "Text field_11" at 38,181 size 17x25; Text 'Text'
   GraphicView "Graphic view_1" at 621,5 size 174x31; Picture "LOGO CREMINOX (1)"
   TextField "Text field_21" at 71,11 size 59x20; Text 'MANUAL'
   Button "Button_17" at 13,0 size 45x40; TextOff 'Text'; PictureOff "Graphic_3"
      on Click: function_efd93a16()
   TextField "Text field_8" at 567,93 size 89x27; Text 'SALIDAS'
   TextField "Text field_9" at 70,93 size 110x27; Text 'ENTRADAS'
   Button "Button_30" at 146,4 size 121x32; TextOff 'CONFIGURACION'
      on Click: ActivateScreen("MENU", 0)
   Button "Button_26" at 279,4 size 102x32; TextOff 'RECETARIO'
      on Click: ActivateScreen("C RECETAS", 0)
      on Release: ResetBit("HMI RECETARIO")
      on Press: SetBit("HMI RECETARIO")
   TextField "Text field_13" at 41,137 size 185x22; Text 'GUARDAMOTOR BOMBA'
      Visibility <- "TIPO DE EQUIPO SELECCIONADO"
   TextField "Text field_14" at 52,172 size 174x22; Text 'SERPENTINA ABIERTA'
      Visibility <- "TIPO DE EQUIPO SELECCIONADO"
   TextField "Text field_15" at 46,210 size 180x22; Text 'SERPENTINA CERRADA'
      Visibility <- "TIPO DE EQUIPO SELECCIONADO"
   TextField "Text field_16" at 53,245 size 173x22; Text 'VAPOR VIVO ABIERTO'
      Visibility <- "TIPO DE EQUIPO SELECCIONADO"
   TextField "Text field_17" at 47,282 size 179x22; Text 'VAPOR VIVO CERRADO'
      Visibility <- "TIPO DE EQUIPO SELECCIONADO"
   TextField "Text field_10" at 69,317 size 156x22; Text 'PULSADOR REARME'
   Circle "Circle_2" at 254,316 size 30x30
      Appearance <- "PRARM"
   TextField "Text field_12" at 32,355 size 194x22; Text 'PULSADOR EMERGENCIA'
   Circle "Circle_1" at 254,353 size 30x30
      Appearance <- "PEMERG"
   TextField "Text field_7" at 45,403 size 64x22; Text 'BUZZER'
   Button "Button_16" at 155,398 size 71x29; TextOff 'OFF'; TextList "Text_list_1"
      on Release: ResetBit("HMI OFF MANUAL BUZZER")
      on Press: SetBit("HMI OFF MANUAL BUZZER")
      Visibility <- "VISUALIZACIONES HMI_BUZZER"
   Circle "Circle_12" at 254,395 size 30x30
      Appearance <- "VISUALIZACIONES HMI_BUZZER"
   TextField "Text field_18" at 14,440 size 122x22; Text 'LUZ PULSADOR'
   Button "Button_21" at 155,436 size 71x29; TextOff 'OFF'; TextList "Text_list_1"
      on Release: ResetBit("HMI OFF LUZ PS REARME")
      on Press: SetBit("HMI OFF LUZ PS REARME")
      Visibility <- "ENTRADAS Y SALIDAS_LUZ MANUAL PS REARME"
   Circle "Circle_15" at 254,435 size 30x30
      Appearance <- "ENTRADAS Y SALIDAS_LUZ MANUAL PS REARME"
   TextField "Text field_6" at 496,211 size 114x22; Text 'BALIZA VERDE'
   TextField "Text field_5" at 505,172 size 105x22; Text 'BALIZA ROJA'
   Button "Button_13" at 634,169 size 71x29; TextOff 'OFF'; TextList "Text_list_1"
      on Release: ResetBit("HMI OFF MANUAL BALIZA ROJA")
      on Press: SetBit("HMI OFF MANUAL BALIZA ROJA")
      Visibility <- "VISUALIZACIONES HMI_ON/OFF BR"
   Button "Button_14" at 634,208 size 71x29; TextOff 'OFF'; TextList "Text_list_1"
      on Release: ResetBit("HMI OFF MANUAL BALIZA VERDE")
      on Press: SetBit("HMI OFF MANUAL BALIZA VERDE")
      Visibility <- "VISUALIZACIONES HMI_ON/OFF BV"
   Circle "Circle_4" at 721,168 size 30x30
      Appearance <- "VISUALIZACIONES HMI_ON/OFF BR"
   Circle "Circle_3" at 721,207 size 30x30
      Appearance <- "VISUALIZACIONES HMI_ON/OFF BV"
   Button "Button_8" at 155,398 size 71x29; TextOff 'ON'; TextList "Text_list_1"
      on Press: SetBit("HMI ON MANUAL BUZZER")
      on Release: ResetBit("HMI ON MANUAL BUZZER")
      Visibility <- "VISUALIZACIONES HMI_BUZZER"
   Button "Button_20" at 155,436 size 71x29; TextOff 'ON'; TextList "Text_list_1"
      on Release: ResetBit("HMI ON LUZ PS REARME")
      on Press: SetBit("HMI ON LUZ PS REARME")
      Visibility <- "ENTRADAS Y SALIDAS_LUZ MANUAL PS REARME"
   Button "Button_6" at 634,208 size 71x29; TextOff 'ON'; TextList "Text_list_1"
      on Press: SetBit("HMI ON MANUAL BALIZA VERDE")
      on Release: ResetBit("HMI ON MANUAL BALIZA VERDE")
      Visibility <- "VISUALIZACIONES HMI_ON/OFF BV"
   Button "Button_5" at 634,169 size 71x29; TextOff 'ON'; TextList "Text_list_1"
      on Press: SetBit("HMI ON MANUAL BALIZA ROJA")
      on Release: ResetBit("HMI ON MANUAL BALIZA ROJA")
      Visibility <- "VISUALIZACIONES HMI_ON/OFF BR"
   TextField "Text field_19" at 500,250 size 110x22; Text 'TOMA FILTRO'
   Button "Button_15" at 634,246 size 71x29; TextOff 'OFF'; TextList "Text_list_1"
      on Release: ResetBit("HMI OFF MANUAL TOMA FILTRO")
      on Press: SetBit("HMI OFF MANUAL TOMA FILTRO")
      Visibility <- "VISUALIZACIONES HMI_ON/OFF TOMA FILTRO"
   Circle "Circle_16" at 721,245 size 30x30
      Appearance <- "VISUALIZACIONES HMI_ON/OFF TOMA FILTRO"
   Button "Button_7" at 634,246 size 71x29; TextOff 'ON'; TextList "Text_list_1"
      on Press: SetBit("HMI ON MANUAL TOMA FILTRO")
      on Release: ResetBit("HMI ON MANUAL TOMA FILTRO")
      Visibility <- "VISUALIZACIONES HMI_ON/OFF TOMA FILTRO"
   TextField "Text field_3" at 483,134 size 127x22; Text 'CARGA DE AGUA'
   Button "Button_3" at 634,130 size 71x29; TextOff 'ON'; TextList "Text_list_1"
      on Press: SetBit("HMI ON MANUAL CARGA AGUA")
      on Release: ResetBit("HMI ON MANUAL CARGA AGUA")
      Visibility <- "VISUALIZACIONES HMI_ON/OFF CARGA AGUA"
   Circle "Circle_6" at 721,130 size 30x30
      Appearance <- "VISUALIZACIONES HMI_ON/OFF CARGA AGUA"
   Button "Button_11" at 634,130 size 71x29; TextOff 'OFF'; TextList "Text_list_1"
      on Release: ResetBit("HMI OFF MANUAL CARGA AGUA")
      on Press: SetBit("HMI OFF MANUAL CARGA AGUA")
      Visibility <- "VISUALIZACIONES HMI_ON/OFF CARGA AGUA"
   TextField "Text field_4" at 417,289 size 193x22; Text 'BOMBA RECIRCULACION'
   Button "Button_12" at 634,284 size 71x29; TextOff 'OFF'; TextList "Text_list_1"
      on Release: ResetBit("HMI OFF MANUAL BOMBA RECIRCULACION")
      on Press: SetBit("HMI OFF MANUAL BOMBA RECIRCULACION")
      Visibility <- "VISUALIZACIONES HMI_ON BOMBA RECIRCULACION"
   Button "Button_4" at 634,284 size 71x29; TextOff 'ON'; TextList "Text_list_1"
      on Press: SetBit("HMI ON MANUAL BOMBA RECIRCULACION")
      on Release: ResetBit("HMI ON MANUAL BOMBA RECIRCULACION")
      Visibility <- "VISUALIZACIONES HMI_ON BOMBA RECIRCULACION"
   Circle "Circle_5" at 721,283 size 30x30
      Appearance <- "VISUALIZACIONES HMI_ON BOMBA RECIRCULACION"
   Circle "Circle_13" at 721,439 size 30x30
      Visibility <- "TIPO DE EQUIPO SELECCIONADO"
      Appearance <- "VISUALIZACIONES HMI_OFF VV"
   Circle "Circle_14" at 721,400 size 30x30
      Visibility <- "TIPO DE EQUIPO SELECCIONADO"
      Appearance <- "VISUALIZACIONES HMI_OFF VS"
   Circle "Circle_7" at 255,133 size 30x30
      Appearance <- "VISUALIZACIONES HMI_GUARDAMOTOR"
      Visibility <- "TIPO DE EQUIPO SELECCIONADO"
   Circle "Circle_8" at 255,168 size 30x30
      Appearance <- "VISUALIZACIONES HMI_SERPENTINA ABIERTA"
      Visibility <- "TIPO DE EQUIPO SELECCIONADO"
   Circle "Circle_9" at 255,206 size 30x30
      Appearance <- "VISUALIZACIONES HMI_SERPENTINA CERRADA"
      Visibility <- "TIPO DE EQUIPO SELECCIONADO"
   Circle "Circle_10" at 255,242 size 30x30
      Appearance <- "VISUALIZACIONES HMI_VAPOR VIVO ABIERTO"
      Visibility <- "TIPO DE EQUIPO SELECCIONADO"
   Circle "Circle_11" at 255,280 size 30x30
      Appearance <- "VISUALIZACIONES HMI_VAPOR VIVO CERRADO"
      Visibility <- "TIPO DE EQUIPO SELECCIONADO"
   Circle "Circle_17" at 721,321 size 30x30
      Visibility <- "TIPO DE EQUIPO SELECCIONADO"
   Circle "Circle_18" at 721,361 size 30x30
      Visibility <- "TIPO DE EQUIPO SELECCIONADO"
   Button "Button_1" at 634,401 size 71x29; TextOff 'ON'; TextList "Text_list_1"
      on Press: SetBit("HMI ON MANUAL VS")
      on Release: ResetBit("HMI ON MANUAL VS")
      Visibility <- "VISUALIZACIONES HMI_ON VS"
   Button "Button_2" at 634,440 size 71x29; TextOff 'ON'; TextList "Text_list_1"
      on Press: SetBit("HMI ON MANUAL VV")
      on Release: ResetBit("HMI ON MANUAL VV")
      Visibility <- "VISUALIZACIONES HMI_ON VV"
   Button "Button_22" at 634,321 size 71x29; TextOff 'ON'; TextList "Text_list_1"
      Visibility <- "VISUALIZACIONES HMI_ON SUBIR TAPA"
      on Press: SetBit("HMI ON LEVANTAR TAPA")
      on Release: ResetBit("HMI ON LEVANTAR TAPA")
   Button "Button_28" at 634,361 size 71x29; TextOff 'ON'; TextList "Text_list_1"
      Visibility <- "VISUALIZACIONES HMI_ON BAJAR TAPA"
      on Press: SetBit("HMI ON BAJAR TAPA")
      on Release: ResetBit("HMI ON BAJAR TAPA")
   Button "Button_9" at 634,401 size 71x29; TextOff 'OFF'; TextList "Text_list_1"
      on Release: ResetBit("HMI OFF MANUAL VS")
      on Press: SetBit("HMI OFF MANUAL VS")
      Visibility <- "VISUALIZACIONES HMI_OFF VS"
   Button "Button_10" at 634,440 size 71x29; TextOff 'OFF'; TextList "Text_list_1"
      on Release: ResetBit("HMI OFF MANUAL VV")
      on Press: SetBit("HMI OFF MANUAL VV")
      Visibility <- "VISUALIZACIONES HMI_OFF VV"
   Button "Button_24" at 634,322 size 71x29; TextOff 'OFF'; TextList "Text_list_1"
      Visibility <- "VISUALIZACIONES HMI_OFF SUBIR TAPA"
      on Press: SetBit("HMI OFF LEVANTAR TAPA")
      on Release: ResetBit("HMI OFF LEVANTAR TAPA")
   Button "Button_31" at 634,362 size 71x29; TextOff 'OFF'; TextList "Text_list_1"
      Visibility <- "VISUALIZACIONES HMI_OFF BAJAR TAPA"
      on Press: SetBit("HMI OFF BAJAR TAPA")
      on Release: ResetBit("HMI OFF BAJAR TAPA")
   TextField "Text field_22" at 93,161 size 122x22; Text 'FALLA CHILLER'
      Visibility <- "TIPO DE EQUIPO SELECCIONADO"
   TextField "Text field_27" at 30,206 size 185x22; Text 'GUARDAMOTOR BOMBA'
      Visibility <- "TIPO DE EQUIPO SELECCIONADO"
   Circle "Circle_22" at 255,157 size 30x30
      Visibility <- "TIPO DE EQUIPO SELECCIONADO"
   Circle "Circle_21" at 255,202 size 30x30
      Visibility <- "TIPO DE EQUIPO SELECCIONADO"
   Circle "Circle_19" at 721,326 size 30x30
      Appearance <- "VISUALIZACIONES HMI_OFF INGRESO AMONIACO"
      Visibility <- "TIPO DE EQUIPO SELECCIONADO"
   TextField "Text field_31" at 494,331 size 114x22; Text 'EV AMONIACO'
      Visibility <- "TIPO DE EQUIPO SELECCIONADO"
   Button "Button_25" at 633,328 size 71x29; TextOff 'ON'; TextList "Text_list_1"
      on Press: SetBit("HMI ON INGRESO AMONIACO")
      on Release: ResetBit("HMI ON INGRESO AMONIACO")
      Visibility <- "VISUALIZACIONES HMI_ON INGRESO AMONIACO"
   Button "Button_29" at 633,328 size 71x29; TextOff 'OFF'; TextList "Text_list_1"
      on Press: SetBit("HMI OFF INGRESO AMONIACO")
      on Release: ResetBit("HMI OFF INGRESO AMONIACO")
      Visibility <- "VISUALIZACIONES HMI_OFF INGRESO AMONIACO"
   Rectangle "Rectangle_2" at 7,89 size 786x384
      Visibility <- "ESTRUCTURAS Y ARREGLOS_HMI ESTADO_EN CICLO"
   IOField "I/O field_16" at 166,49 size 215x35; FormatPattern ??????????????????????????
      ProcessValue <- "ESTRUCTURAS Y ARREGLOS_HMI NOMBRE EQUIPO"
   Button "Button_19" at 400,49 size 39x35; TextOff 'Text'; PictureOff "Graphic_1"
      on Release: ResetBit("HMI DISMINUIR EQUIPO")
      on Press: SetBit("HMI DISMINUIR EQUIPO")
      Visibility <- "VISUALIZACIONES HMI_LIM INF EQUIPO SEL"
   IOField "I/O field_2" at 464,49 size 42x35; FormatPattern 99
      ProcessValue <- "EQUIPO SELECCIONADO"
   Button "Button_18" at 531,49 size 40x35; TextOff 'Text'; PictureOff "Graphic_2"
      on Release: ResetBit("HMI AUMENTAR EQUIPO")
      on Press: SetBit("HMI AUMENTAR EQUIPO")
      Visibility <- "VISUALIZACIONES HMI_LIM SUP EQUIPO SEL"

screen "PRINCIPAL" 800x480
   Rectangle "Rectangle_2" at 401,39 size 398x440
      Appearance <- "ESTRUCTURAS Y ARREGLOS_ESTADO{2}_COLOR EN HMI"
   Rectangle "Rectangle_1" at 2,39 size 400x442
      Appearance <- "ESTRUCTURAS Y ARREGLOS_ESTADO{1}_COLOR EN HMI"
   TextField "Text field_2" at 18,46 size 169x22; Text 'EQUIPO 1 - COCINA 1'
   TextField "Text field_3" at 417,46 size 200x22; Text 'EQUIPO 2 - ENFRIADOR 1'
   TextField "Text field_6" at 27,157 size 37x17; Text 'AGUA'
   TextField "Text field_8" at 164,157 size 57x17; Text 'INGRESO'
   TextField "Text field_9" at 313,157 size 69x17; Text 'PRODUCTO'
   TextField "Text field_10" at 119,73 size 164x22; Text 'ESTADO DEL EQUIPO'
   Button "Button_1" at 18,444 size 359x28; TextOff 'VER EQUIPO'
      on Click: ActivateScreen("EQUIPO", 0)
      on Press: SetBit("HMI VER EQUIPO 1")
      on Release: ResetBit("HMI VER EQUIPO 1")
   Button "Button_2" at 18,409 size 359x28; TextOff 'GRAFICO TEMPERATURAS'
      on Press: SetBit("HMI VER EQUIPO 1")
      on Release: ResetBit("HMI VER EQUIPO 1")
      on Click: ActivateScreen("GRAFICOS", 0)
   TextField "Text field_14" at 442,157 size 40x17; Text 'AGUA'
   TextField "Text field_16" at 566,157 size 54x17; Text 'INGRESO'
   TextField "Text field_17" at 709,157 size 66x17; Text 'PRODUCTO'
   Button "Button_3" at 425,444 size 362x28; TextOff 'VER EQUIPO'
      on Click: ActivateScreen("EQUIPO", 0)
      on Press: SetBit("HMI VER EQUIPO 2")
      on Release: ResetBit("HMI VER EQUIPO 2")
   Button "Button_4" at 425,409 size 362x28; TextOff 'GRAFICO TEMPERATURAS'
      on Press: SetBit("HMI VER EQUIPO 2")
      on Release: ResetBit("HMI VER EQUIPO 2")
      on Click: ActivateScreen("GRAFICOS", 0)
   TextField "Text field_20" at 416,374 size 155x20; Text 'TIEMPO TRANSCURRIDO'
   TextField "Text field_38" at 228,0 size 17x25; Text 'Text'
   IOField "I/O field_1" at 11,180 size 74x25; FormatPattern 99.9; Unit  °C
      ProcessValue <- "ESTRUCTURAS Y ARREGLOS_TEMPERATURAS{1}_TEMPERATURA AGUA"
   IOField "I/O field_2" at 156,180 size 76x26; FormatPattern 99.9; Unit  °C
      ProcessValue <- "ESTRUCTURAS Y ARREGLOS_TEMPERATURAS{1}_TEMPERATURA INGRESO"
   IOField "I/O field_3" at 303,179 size 84x27; FormatPattern 99.9; Unit  °C
      ProcessValue <- "ESTRUCTURAS Y ARREGLOS_TEMPERATURAS{1}_TEMPERATURA PRODUCTO"
   IOField "I/O field_4" at 79,215 size 85x26; FormatPattern 9999; Unit  mm
      ProcessValue <- "ESTRUCTURAS Y ARREGLOS_NIVEL{1}"
   IOField "I/O field_5" at 332,215 size 27x27; FormatPattern 9
      ProcessValue <- "ESTRUCTURAS Y ARREGLOS_CARGA{1}_CANTIDAD DE TORRES"
   IOField "I/O field_7" at 11,99 size 380x26; FormatPattern ????????????????????????????
      ProcessValue <- "ESTRUCTURAS Y ARREGLOS_ESTADO{1}_EQUIPO"
   IOField "I/O field_8" at 179,376 size 72x25; FormatPattern 999; Unit  min
      ProcessValue <- "ESTRUCTURAS Y ARREGLOS_ESTADO{1}_TIEMPO TRANSCURRIDO"
   IOField "I/O field_9" at 408,99 size 384x27; FormatPattern ????????????????????????????
      ProcessValue <- "ESTRUCTURAS Y ARREGLOS_ESTADO{2}_EQUIPO"
   IOField "I/O field_10" at 412,179 size 84x27; FormatPattern 99.9; Unit  °C
      ProcessValue <- "ESTRUCTURAS Y ARREGLOS_TEMPERATURAS{2}_TEMPERATURA AGUA"
   IOField "I/O field_11" at 552,179 size 85x27; FormatPattern 99.9; Unit  °C
      ProcessValue <- "ESTRUCTURAS Y ARREGLOS_TEMPERATURAS{2}_TEMPERATURA INGRESO"
   IOField "I/O field_12" at 700,179 size 85x27; FormatPattern 99.9; Unit  °C
      ProcessValue <- "ESTRUCTURAS Y ARREGLOS_TEMPERATURAS{2}_TEMPERATURA PRODUCTO"
   IOField "I/O field_13" at 480,215 size 84x26; FormatPattern 9999; Unit  mm
      ProcessValue <- "ESTRUCTURAS Y ARREGLOS_NIVEL{2}"
   IOField "I/O field_14" at 725,215 size 25x27; FormatPattern 9
      ProcessValue <- "ESTRUCTURAS Y ARREGLOS_CARGA{2}_CANTIDAD DE TORRES"
   IOField "I/O field_15" at 411,308 size 381x27; FormatPattern ?????????????????????????
      ProcessValue <- "ESTRUCTURAS Y ARREGLOS_CARGA RECETA{2}_NOMBRE"
   IOField "I/O field_16" at 582,371 size 72x25; FormatPattern 999; Unit  min
      ProcessValue <- "ESTRUCTURAS Y ARREGLOS_ESTADO{2}_TIEMPO TRANSCURRIDO"
   IOField "I/O field_6" at 18,308 size 372x26; FormatPattern ?????????????????????????
      ProcessValue <- "ESTRUCTURAS Y ARREGLOS_CARGA RECETA{1}_NOMBRE"
   Button "Button_11" at 4,3 size 96x32; TextOff 'MANUAL'
      on Click: ActivateScreen("MANUAL", 0)
   Button "Button_12" at 103,3 size 121x32; TextOff 'CONFIGURACION'
      on Click: ActivateScreen("MENU", 0)
   Button "Button_26" at 332,4 size 116x32; TextOff 'CERRAR SESION'
      on Click: function_f23ef4c9()
   Button "Button_13" at 226,3 size 102x32; TextOff 'RECETARIO'
      on Click: ActivateScreen("C RECETAS", 0)
      on Press: SetBit("HMI RECETARIO")
      on Release: ResetBit("HMI RECETARIO")
   TextField "Text field_1" at 518,72 size 164x22; Text 'ESTADO DEL EQUIPO'
   TextField "Text field_5" at 637,217 size 67x22; Text 'TORRES'
   TextField "Text field_15" at 416,217 size 52x22; Text 'NIVEL'
   TextField "Text field_18" at 509,279 size 186x22; Text 'RECETA SELECCIONADA'
   TextField "Text field_21" at 245,217 size 67x22; Text 'TORRES'
   TextField "Text field_7" at 11,217 size 52x22; Text 'NIVEL'
   TextField "Text field_11" at 109,279 size 186x22; Text 'RECETA SELECCIONADA'
   TextField "Text field_12" at 12,378 size 155x20; Text 'TIEMPO TRANSCURRIDO'
   IOField "I/O field_17" at 129,344 size 39x29; FormatPattern 99
      ProcessValue <- "ESTRUCTURAS Y ARREGLOS_HMI ESTADO_PASO ACTUAL"
      Visibility <- "VISUALIZACIONES HMI_PASOS OP EN COCINAS"
   TextField "Text field_13" at 12,347 size 98x20; Text 'PASO ACTUAL'
      Visibility <- "VISUALIZACIONES HMI_PASOS OP EN COCINAS"
   TextField "Text field_22" at 12,252 size 44x22; Text 'LOTE'
   IOField "I/O field_18" at 79,249 size 249x26; FormatPattern 9999999
   TextField "Text field_4" at 138,130 size 127x22; Text 'TEMPERATURAS'
   TextField "Text field_19" at 537,130 size 127x22; Text 'TEMPERATURAS'
   TextField "Text field_23" at 418,252 size 44x22; Text 'LOTE'
   IOField "I/O field_19" at 480,249 size 249x26; FormatPattern 9999999
   GraphicView "Graphic view_1" at 628,4 size 174x31; Picture "LOGO CREMINOX (1)"

